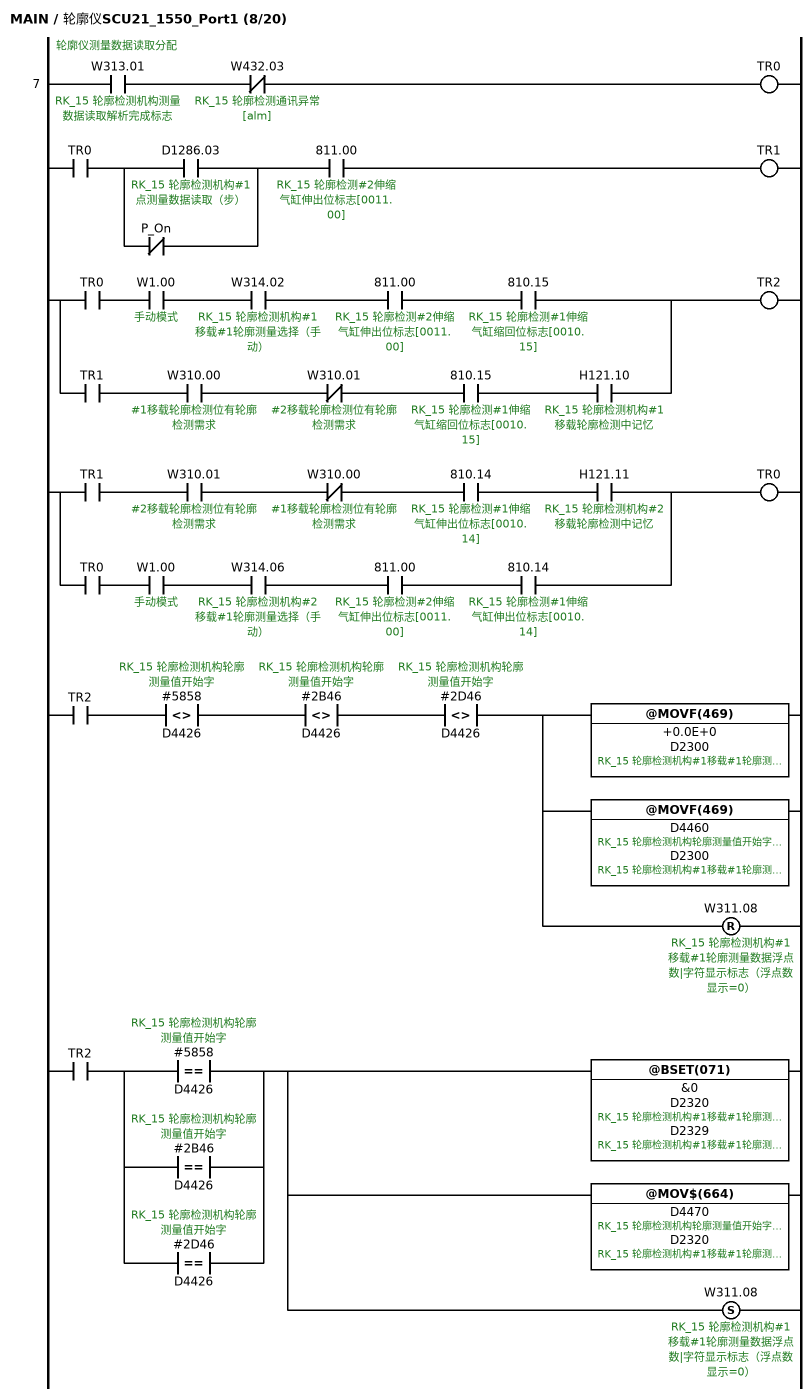
; [picture p24: MAIN / 轮廓仪SCU21_1550_Port1, rungs 7-7]

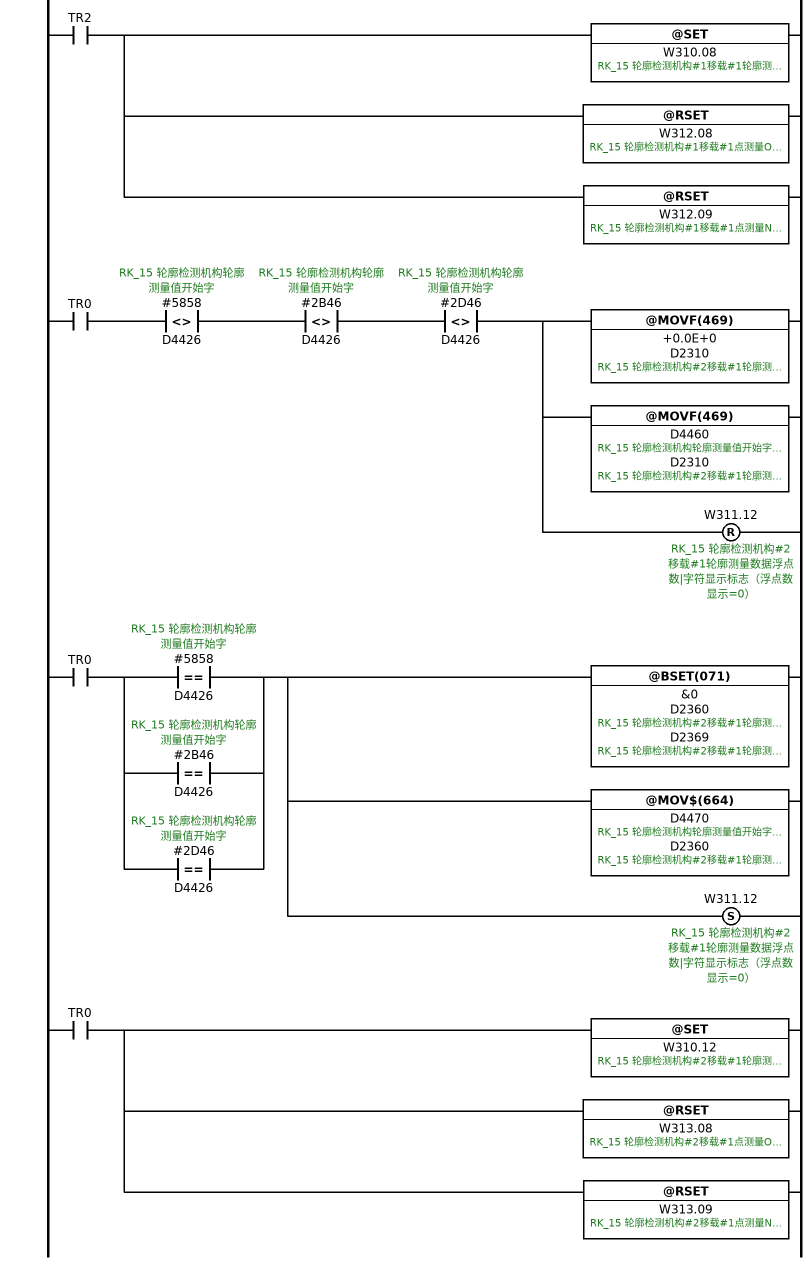
; rung 7: 轮廓仪测量数据读取分配
LD W313.01  ; RK_15 轮廓检测机构测量数据读取解析完成标志
ANDNOT W432.03  ; RK_15 轮廓检测通讯异常[alm]
OUT TR0
AND W1.00  ; 手动模式
AND W314.02  ; RK_15 轮廓检测机构#1移载#1轮廓测量选择（手动）
AND 811.00  ; RK_15 轮廓检测#2伸缩气缸伸出位标志[0011.00]
AND 810.15  ; RK_15 轮廓检测#1伸缩气缸缩回位标志[0010.15]
LD TR0
LD D1286.03  ; RK_15 轮廓检测机构#1点测量数据读取（步）
ORNOT P_On
ANDLD
AND 811.00  ; RK_15 轮廓检测#2伸缩气缸伸出位标志[0011.00]
OUT TR1
AND W310.00  ; #1移载轮廓检测位有轮廓检测需求
ANDNOT W310.01  ; #2移载轮廓检测位有轮廓检测需求
AND 810.15  ; RK_15 轮廓检测#1伸缩气缸缩回位标志[0010.15]
AND H121.10  ; RK_15 轮廓检测机构#1移载轮廓检测中记忆
ORLD
OUT TR2
AND<>(305) #5858 D4426  ; RK_15 轮廓检测机构轮廓测量值开始字
AND<>(305) #2B46 D4426  ; RK_15 轮廓检测机构轮廓测量值开始字
AND<>(305) #2D46 D4426  ; RK_15 轮廓检测机构轮廓测量值开始字
@MOVF(469) +0.0E+0 D2300  ; RK_15 轮廓检测机构#1移载#1轮廓测量值（Float）
@MOVF(469) D4460 D2300  ; RK_15 轮廓检测机构轮廓测量值开始字（Float）, RK_15 轮廓检测机构#1移载#1轮廓测量值（Float）
RSET W311.08  ; RK_15 轮廓检测机构#1移载#1轮廓测量数据浮点数|字符显示标志（浮点数显示=0）
LD TR2
LD=(300) #5858 D4426  ; RK_15 轮廓检测机构轮廓测量值开始字
OR=(300) #2B46 D4426  ; RK_15 轮廓检测机构轮廓测量值开始字
OR=(300) #2D46 D4426  ; RK_15 轮廓检测机构轮廓测量值开始字
ANDLD
@BSET(071) &0 D2320 D2329  ; RK_15 轮廓检测机构#1移载#1轮廓测量值开始字（String）, RK_15 轮廓检测机构#1移载#1轮廓测量值结束字（String）
@MOV$(664) D4470 D2320  ; RK_15 轮廓检测机构轮廓测量值开始字（String）, RK_15 轮廓检测机构#1移载#1轮廓测量值开始字（String）
SET W311.08  ; RK_15 轮廓检测机构#1移载#1轮廓测量数据浮点数|字符显示标志（浮点数显示=0）
LD TR2
@SET W310.08  ; RK_15 轮廓检测机构#1移载#1轮廓测量值读取标志
@RSET W312.08  ; RK_15 轮廓检测机构#1移载#1点测量OK标志
@RSET W312.09  ; RK_15 轮廓检测机构#1移载#1点测量NG标志
LD TR1
AND W310.01  ; #2移载轮廓检测位有轮廓检测需求
ANDNOT W310.00  ; #1移载轮廓检测位有轮廓检测需求
AND 810.14  ; RK_15 轮廓检测#1伸缩气缸伸出位标志[0010.14]
AND H121.11  ; RK_15 轮廓检测机构#2移载轮廓检测中记忆
LD TR0
AND W1.00  ; 手动模式
AND W314.06  ; RK_15 轮廓检测机构#2移载#1轮廓测量选择（手动）
AND 811.00  ; RK_15 轮廓检测#2伸缩气缸伸出位标志[0011.00]
AND 810.14  ; RK_15 轮廓检测#1伸缩气缸伸出位标志[0010.14]
ORLD
OUT TR0
AND<>(305) #5858 D4426  ; RK_15 轮廓检测机构轮廓测量值开始字
AND<>(305) #2B46 D4426  ; RK_15 轮廓检测机构轮廓测量值开始字
AND<>(305) #2D46 D4426  ; RK_15 轮廓检测机构轮廓测量值开始字
@MOVF(469) +0.0E+0 D2310  ; RK_15 轮廓检测机构#2移载#1轮廓测量值（Float）
@MOVF(469) D4460 D2310  ; RK_15 轮廓检测机构轮廓测量值开始字（Float）, RK_15 轮廓检测机构#2移载#1轮廓测量值（Float）
RSET W311.12  ; RK_15 轮廓检测机构#2移载#1轮廓测量数据浮点数|字符显示标志（浮点数显示=0）
LD TR0
LD=(300) #5858 D4426  ; RK_15 轮廓检测机构轮廓测量值开始字
OR=(300) #2B46 D4426  ; RK_15 轮廓检测机构轮廓测量值开始字
OR=(300) #2D46 D4426  ; RK_15 轮廓检测机构轮廓测量值开始字
ANDLD
@BSET(071) &0 D2360 D2369  ; RK_15 轮廓检测机构#2移载#1轮廓测量值开始字（String）, RK_15 轮廓检测机构#2移载#1轮廓测量值结束字（String）
@MOV$(664) D4470 D2360  ; RK_15 轮廓检测机构轮廓测量值开始字（String）, RK_15 轮廓检测机构#2移载#1轮廓测量值开始字（String）
SET W311.12  ; RK_15 轮廓检测机构#2移载#1轮廓测量数据浮点数|字符显示标志（浮点数显示=0）
LD TR0
@SET W310.12  ; RK_15 轮廓检测机构#2移载#1轮廓测量值读取标志
@RSET W313.08  ; RK_15 轮廓检测机构#2移载#1点测量OK标志
@RSET W313.09  ; RK_15 轮廓检测机构#2移载#1点测量NG标志

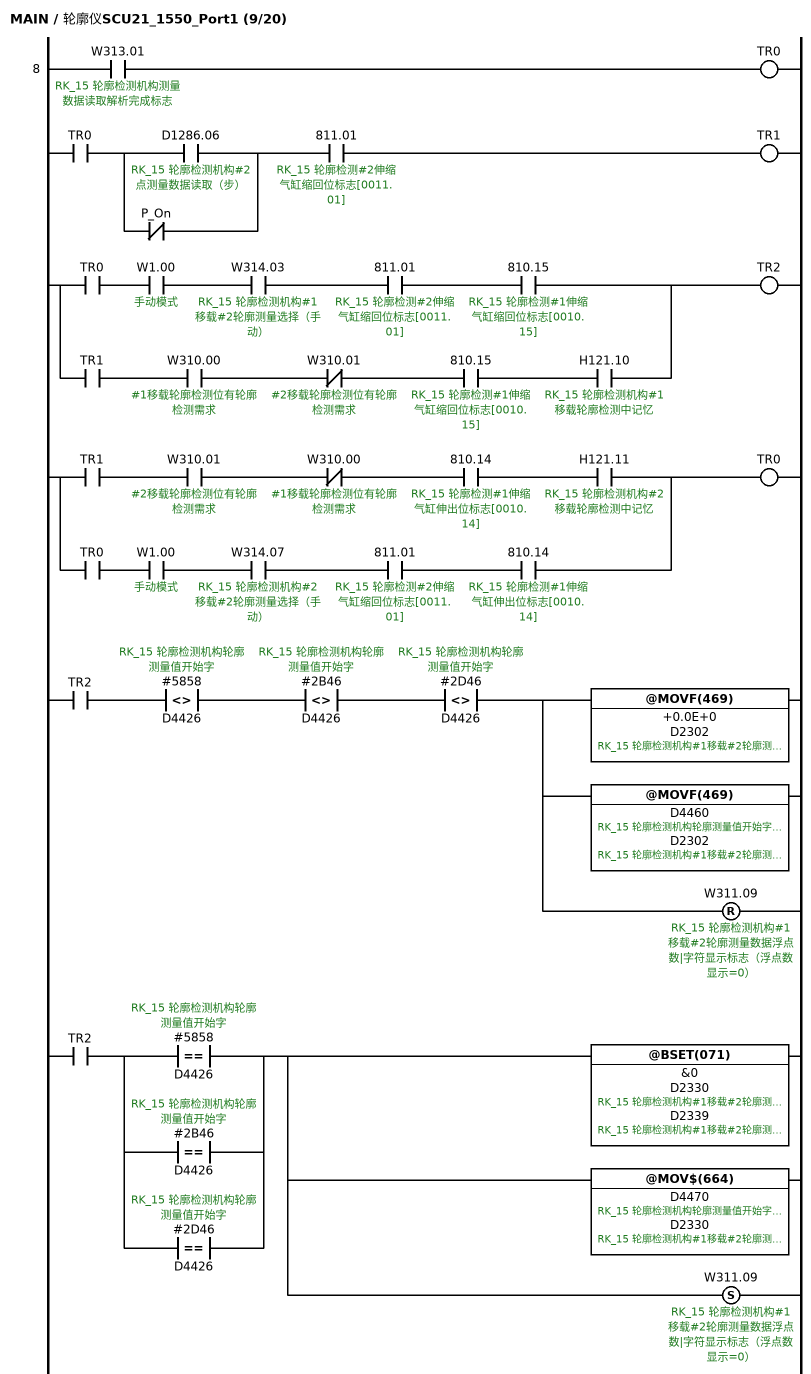

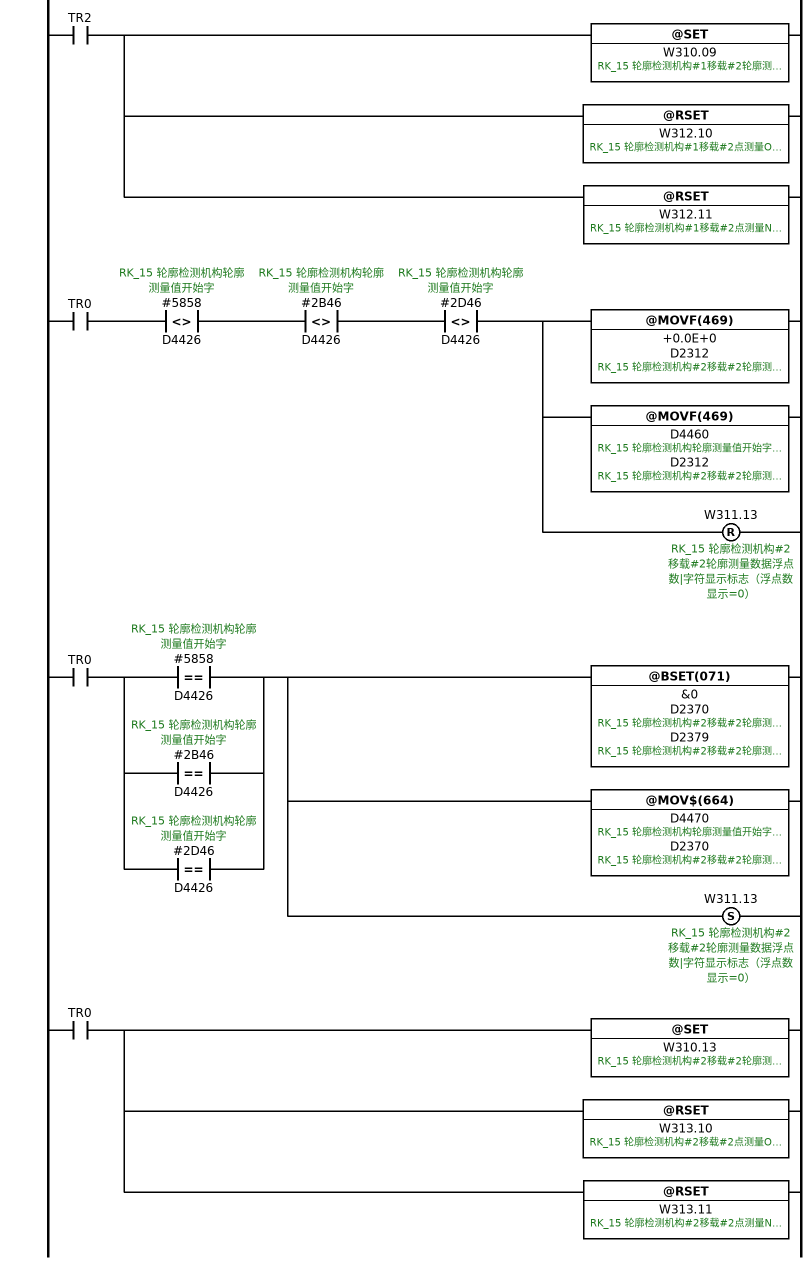
; rung 8
LD W313.01  ; RK_15 轮廓检测机构测量数据读取解析完成标志
OUT TR0
AND W1.00  ; 手动模式
AND W314.03  ; RK_15 轮廓检测机构#1移载#2轮廓测量选择（手动）
AND 811.01  ; RK_15 轮廓检测#2伸缩气缸缩回位标志[0011.01]
AND 810.15  ; RK_15 轮廓检测#1伸缩气缸缩回位标志[0010.15]
LD TR0
LD D1286.06  ; RK_15 轮廓检测机构#2点测量数据读取（步）
ORNOT P_On
ANDLD
AND 811.01  ; RK_15 轮廓检测#2伸缩气缸缩回位标志[0011.01]
OUT TR1
AND W310.00  ; #1移载轮廓检测位有轮廓检测需求
ANDNOT W310.01  ; #2移载轮廓检测位有轮廓检测需求
AND 810.15  ; RK_15 轮廓检测#1伸缩气缸缩回位标志[0010.15]
AND H121.10  ; RK_15 轮廓检测机构#1移载轮廓检测中记忆
ORLD
OUT TR2
AND<>(305) #5858 D4426  ; RK_15 轮廓检测机构轮廓测量值开始字
AND<>(305) #2B46 D4426  ; RK_15 轮廓检测机构轮廓测量值开始字
AND<>(305) #2D46 D4426  ; RK_15 轮廓检测机构轮廓测量值开始字
@MOVF(469) +0.0E+0 D2302  ; RK_15 轮廓检测机构#1移载#2轮廓测量值（Float）
@MOVF(469) D4460 D2302  ; RK_15 轮廓检测机构轮廓测量值开始字（Float）, RK_15 轮廓检测机构#1移载#2轮廓测量值（Float）
RSET W311.09  ; RK_15 轮廓检测机构#1移载#2轮廓测量数据浮点数|字符显示标志（浮点数显示=0）
LD TR2
LD=(300) #5858 D4426  ; RK_15 轮廓检测机构轮廓测量值开始字
OR=(300) #2B46 D4426  ; RK_15 轮廓检测机构轮廓测量值开始字
OR=(300) #2D46 D4426  ; RK_15 轮廓检测机构轮廓测量值开始字
ANDLD
@BSET(071) &0 D2330 D2339  ; RK_15 轮廓检测机构#1移载#2轮廓测量值开始字（String）, RK_15 轮廓检测机构#1移载#2轮廓测量值结束字（String）
@MOV$(664) D4470 D2330  ; RK_15 轮廓检测机构轮廓测量值开始字（String）, RK_15 轮廓检测机构#1移载#2轮廓测量值开始字（String）
SET W311.09  ; RK_15 轮廓检测机构#1移载#2轮廓测量数据浮点数|字符显示标志（浮点数显示=0）
LD TR2
@SET W310.09  ; RK_15 轮廓检测机构#1移载#2轮廓测量值读取标志
@RSET W312.10  ; RK_15 轮廓检测机构#1移载#2点测量OK标志
@RSET W312.11  ; RK_15 轮廓检测机构#1移载#2点测量NG标志
LD TR1
AND W310.01  ; #2移载轮廓检测位有轮廓检测需求
ANDNOT W310.00  ; #1移载轮廓检测位有轮廓检测需求
AND 810.14  ; RK_15 轮廓检测#1伸缩气缸伸出位标志[0010.14]
AND H121.11  ; RK_15 轮廓检测机构#2移载轮廓检测中记忆
LD TR0
AND W1.00  ; 手动模式
AND W314.07  ; RK_15 轮廓检测机构#2移载#2轮廓测量选择（手动）
AND 811.01  ; RK_15 轮廓检测#2伸缩气缸缩回位标志[0011.01]
AND 810.14  ; RK_15 轮廓检测#1伸缩气缸伸出位标志[0010.14]
ORLD
OUT TR0
AND<>(305) #5858 D4426  ; RK_15 轮廓检测机构轮廓测量值开始字
AND<>(305) #2B46 D4426  ; RK_15 轮廓检测机构轮廓测量值开始字
AND<>(305) #2D46 D4426  ; RK_15 轮廓检测机构轮廓测量值开始字
@MOVF(469) +0.0E+0 D2312  ; RK_15 轮廓检测机构#2移载#2轮廓测量值（Float）
@MOVF(469) D4460 D2312  ; RK_15 轮廓检测机构轮廓测量值开始字（Float）, RK_15 轮廓检测机构#2移载#2轮廓测量值（Float）
RSET W311.13  ; RK_15 轮廓检测机构#2移载#2轮廓测量数据浮点数|字符显示标志（浮点数显示=0）
LD TR0
LD=(300) #5858 D4426  ; RK_15 轮廓检测机构轮廓测量值开始字
OR=(300) #2B46 D4426  ; RK_15 轮廓检测机构轮廓测量值开始字
OR=(300) #2D46 D4426  ; RK_15 轮廓检测机构轮廓测量值开始字
ANDLD
@BSET(071) &0 D2370 D2379  ; RK_15 轮廓检测机构#2移载#2轮廓测量值开始字（String）, RK_15 轮廓检测机构#2移载#2轮廓测量值结束字（String）
@MOV$(664) D4470 D2370  ; RK_15 轮廓检测机构轮廓测量值开始字（String）, RK_15 轮廓检测机构#2移载#2轮廓测量值开始字（String）
SET W311.13  ; RK_15 轮廓检测机构#2移载#2轮廓测量数据浮点数|字符显示标志（浮点数显示=0）
LD TR0
@SET W310.13  ; RK_15 轮廓检测机构#2移载#2轮廓测量值读取标志
@RSET W313.10  ; RK_15 轮廓检测机构#2移载#2点测量OK标志
@RSET W313.11  ; RK_15 轮廓检测机构#2移载#2点测量NG标志

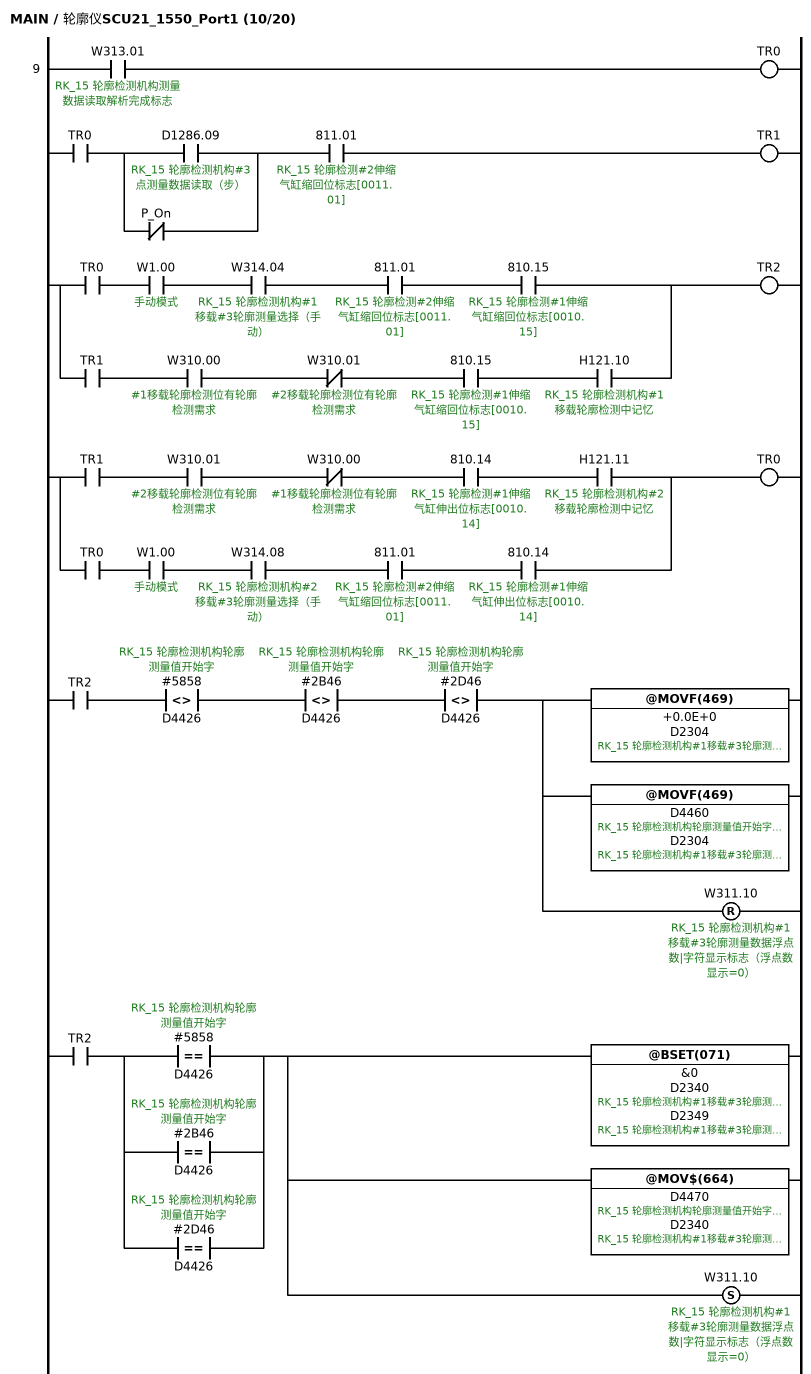

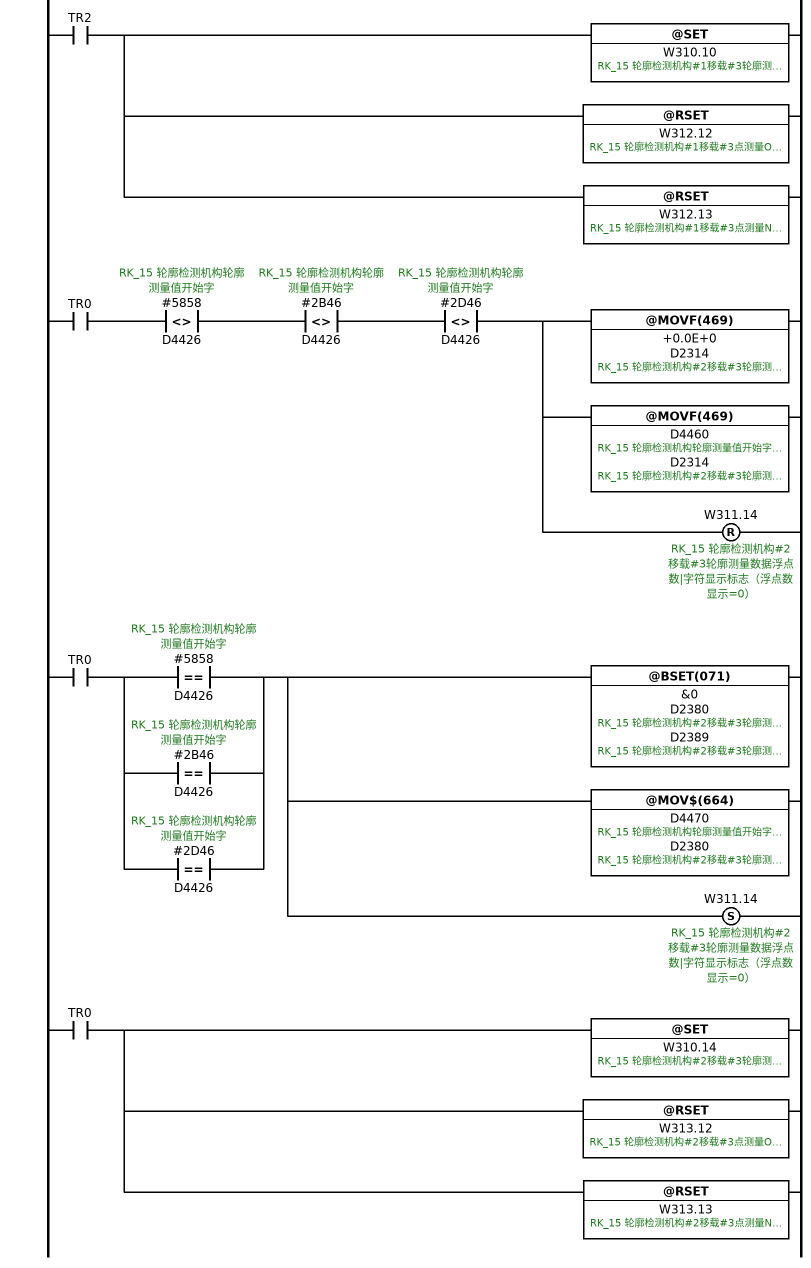
; rung 9
LD W313.01  ; RK_15 轮廓检测机构测量数据读取解析完成标志
OUT TR0
AND W1.00  ; 手动模式
AND W314.04  ; RK_15 轮廓检测机构#1移载#3轮廓测量选择（手动）
AND 811.01  ; RK_15 轮廓检测#2伸缩气缸缩回位标志[0011.01]
AND 810.15  ; RK_15 轮廓检测#1伸缩气缸缩回位标志[0010.15]
LD TR0
LD D1286.09  ; RK_15 轮廓检测机构#3点测量数据读取（步）
ORNOT P_On
ANDLD
AND 811.01  ; RK_15 轮廓检测#2伸缩气缸缩回位标志[0011.01]
OUT TR1
AND W310.00  ; #1移载轮廓检测位有轮廓检测需求
ANDNOT W310.01  ; #2移载轮廓检测位有轮廓检测需求
AND 810.15  ; RK_15 轮廓检测#1伸缩气缸缩回位标志[0010.15]
AND H121.10  ; RK_15 轮廓检测机构#1移载轮廓检测中记忆
ORLD
OUT TR2
AND<>(305) #5858 D4426  ; RK_15 轮廓检测机构轮廓测量值开始字
AND<>(305) #2B46 D4426  ; RK_15 轮廓检测机构轮廓测量值开始字
AND<>(305) #2D46 D4426  ; RK_15 轮廓检测机构轮廓测量值开始字
@MOVF(469) +0.0E+0 D2304  ; RK_15 轮廓检测机构#1移载#3轮廓测量值（Float）
@MOVF(469) D4460 D2304  ; RK_15 轮廓检测机构轮廓测量值开始字（Float）, RK_15 轮廓检测机构#1移载#3轮廓测量值（Float）
RSET W311.10  ; RK_15 轮廓检测机构#1移载#3轮廓测量数据浮点数|字符显示标志（浮点数显示=0）
LD TR2
LD=(300) #5858 D4426  ; RK_15 轮廓检测机构轮廓测量值开始字
OR=(300) #2B46 D4426  ; RK_15 轮廓检测机构轮廓测量值开始字
OR=(300) #2D46 D4426  ; RK_15 轮廓检测机构轮廓测量值开始字
ANDLD
@BSET(071) &0 D2340 D2349  ; RK_15 轮廓检测机构#1移载#3轮廓测量值开始字（String）, RK_15 轮廓检测机构#1移载#3轮廓测量值结束字（String）
@MOV$(664) D4470 D2340  ; RK_15 轮廓检测机构轮廓测量值开始字（String）, RK_15 轮廓检测机构#1移载#3轮廓测量值开始字（String）
SET W311.10  ; RK_15 轮廓检测机构#1移载#3轮廓测量数据浮点数|字符显示标志（浮点数显示=0）
LD TR2
@SET W310.10  ; RK_15 轮廓检测机构#1移载#3轮廓测量值读取标志
@RSET W312.12  ; RK_15 轮廓检测机构#1移载#3点测量OK标志
@RSET W312.13  ; RK_15 轮廓检测机构#1移载#3点测量NG标志
LD TR1
AND W310.01  ; #2移载轮廓检测位有轮廓检测需求
ANDNOT W310.00  ; #1移载轮廓检测位有轮廓检测需求
AND 810.14  ; RK_15 轮廓检测#1伸缩气缸伸出位标志[0010.14]
AND H121.11  ; RK_15 轮廓检测机构#2移载轮廓检测中记忆
LD TR0
AND W1.00  ; 手动模式
AND W314.08  ; RK_15 轮廓检测机构#2移载#3轮廓测量选择（手动）
AND 811.01  ; RK_15 轮廓检测#2伸缩气缸缩回位标志[0011.01]
AND 810.14  ; RK_15 轮廓检测#1伸缩气缸伸出位标志[0010.14]
ORLD
OUT TR0
AND<>(305) #5858 D4426  ; RK_15 轮廓检测机构轮廓测量值开始字
AND<>(305) #2B46 D4426  ; RK_15 轮廓检测机构轮廓测量值开始字
AND<>(305) #2D46 D4426  ; RK_15 轮廓检测机构轮廓测量值开始字
@MOVF(469) +0.0E+0 D2314  ; RK_15 轮廓检测机构#2移载#3轮廓测量值（Float）
@MOVF(469) D4460 D2314  ; RK_15 轮廓检测机构轮廓测量值开始字（Float）, RK_15 轮廓检测机构#2移载#3轮廓测量值（Float）
RSET W311.14  ; RK_15 轮廓检测机构#2移载#3轮廓测量数据浮点数|字符显示标志（浮点数显示=0）
LD TR0
LD=(300) #5858 D4426  ; RK_15 轮廓检测机构轮廓测量值开始字
OR=(300) #2B46 D4426  ; RK_15 轮廓检测机构轮廓测量值开始字
OR=(300) #2D46 D4426  ; RK_15 轮廓检测机构轮廓测量值开始字
ANDLD
@BSET(071) &0 D2380 D2389  ; RK_15 轮廓检测机构#2移载#3轮廓测量值开始字（String）, RK_15 轮廓检测机构#2移载#3轮廓测量值结束字（String）
@MOV$(664) D4470 D2380  ; RK_15 轮廓检测机构轮廓测量值开始字（String）, RK_15 轮廓检测机构#2移载#3轮廓测量值开始字（String）
SET W311.14  ; RK_15 轮廓检测机构#2移载#3轮廓测量数据浮点数|字符显示标志（浮点数显示=0）
LD TR0
@SET W310.14  ; RK_15 轮廓检测机构#2移载#3轮廓测量值读取标志
@RSET W313.12  ; RK_15 轮廓检测机构#2移载#3点测量OK标志
@RSET W313.13  ; RK_15 轮廓检测机构#2移载#3点测量NG标志

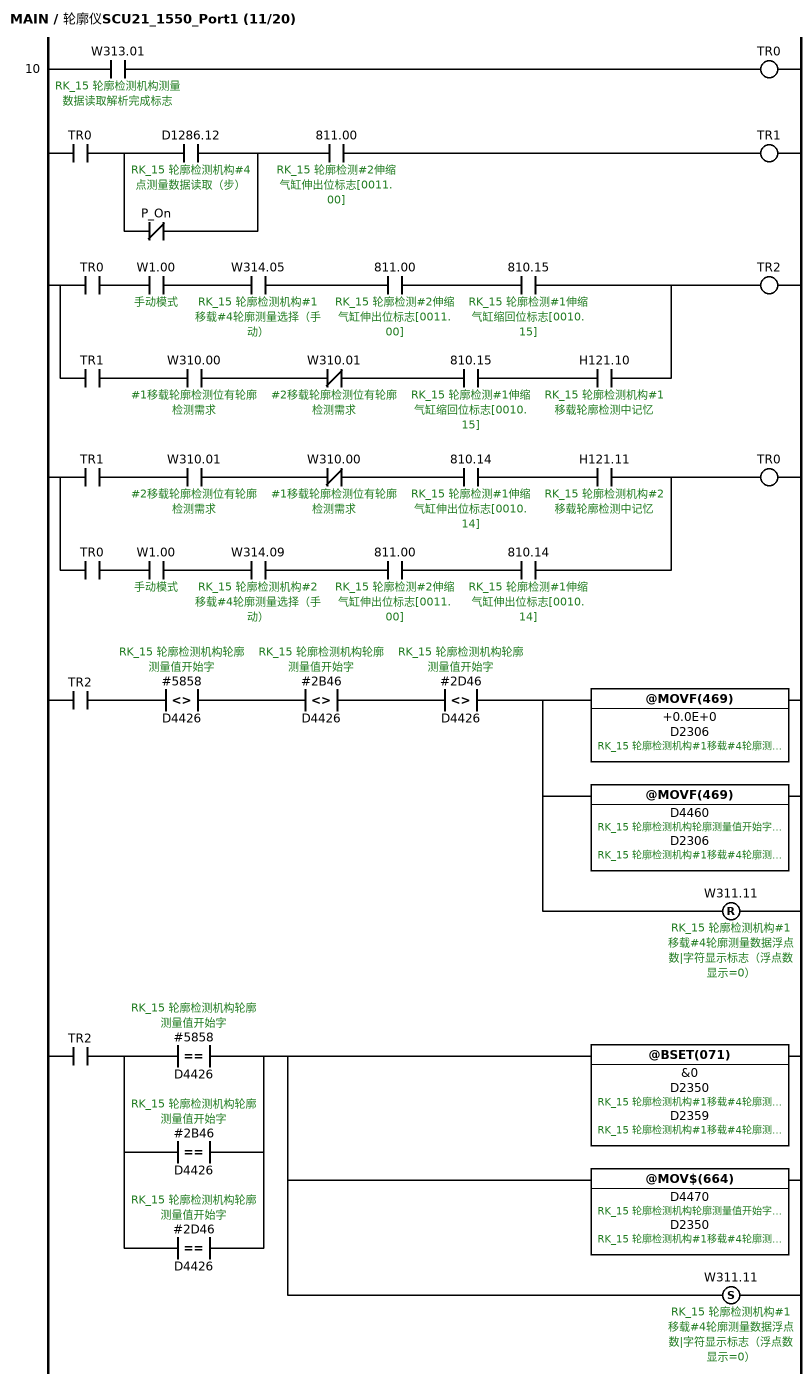

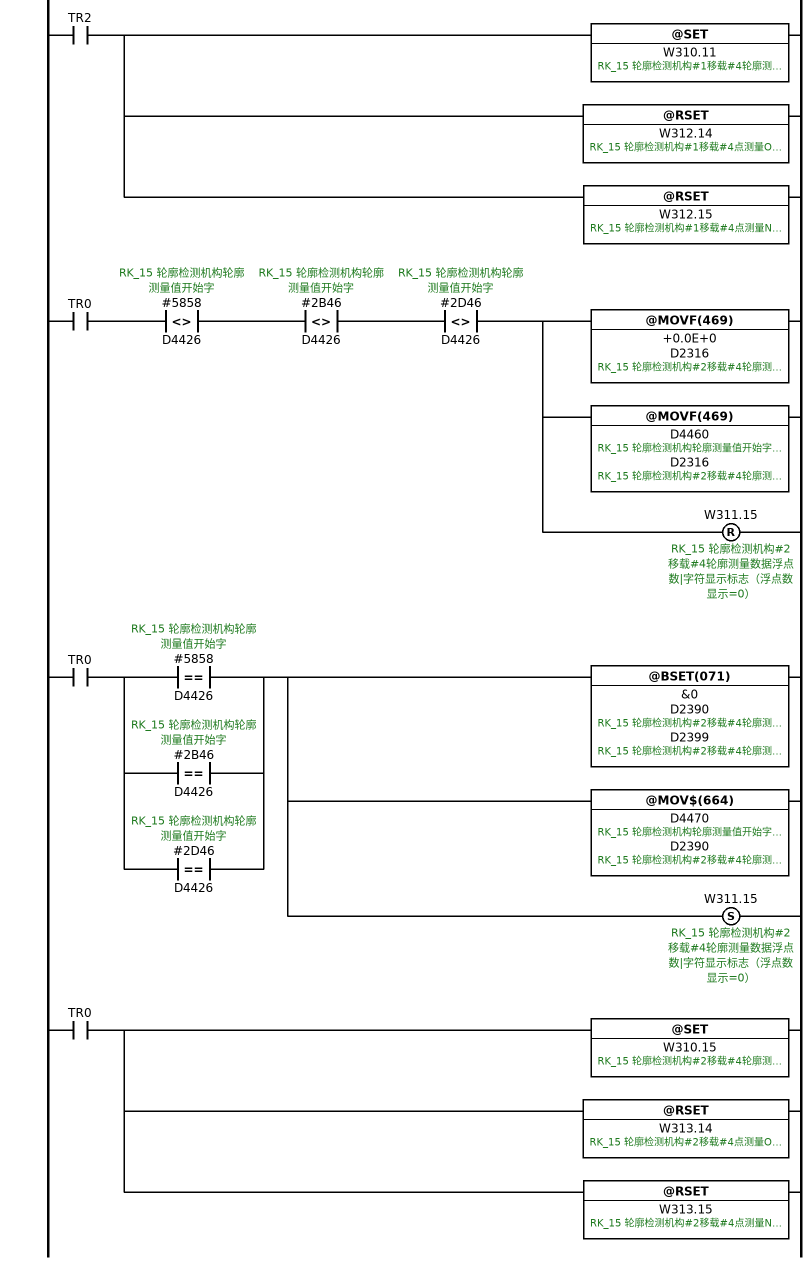
; rung 10
LD W313.01  ; RK_15 轮廓检测机构测量数据读取解析完成标志
OUT TR0
AND W1.00  ; 手动模式
AND W314.05  ; RK_15 轮廓检测机构#1移载#4轮廓测量选择（手动）
AND 811.00  ; RK_15 轮廓检测#2伸缩气缸伸出位标志[0011.00]
AND 810.15  ; RK_15 轮廓检测#1伸缩气缸缩回位标志[0010.15]
LD TR0
LD D1286.12  ; RK_15 轮廓检测机构#4点测量数据读取（步）
ORNOT P_On
ANDLD
AND 811.00  ; RK_15 轮廓检测#2伸缩气缸伸出位标志[0011.00]
OUT TR1
AND W310.00  ; #1移载轮廓检测位有轮廓检测需求
ANDNOT W310.01  ; #2移载轮廓检测位有轮廓检测需求
AND 810.15  ; RK_15 轮廓检测#1伸缩气缸缩回位标志[0010.15]
AND H121.10  ; RK_15 轮廓检测机构#1移载轮廓检测中记忆
ORLD
OUT TR2
AND<>(305) #5858 D4426  ; RK_15 轮廓检测机构轮廓测量值开始字
AND<>(305) #2B46 D4426  ; RK_15 轮廓检测机构轮廓测量值开始字
AND<>(305) #2D46 D4426  ; RK_15 轮廓检测机构轮廓测量值开始字
@MOVF(469) +0.0E+0 D2306  ; RK_15 轮廓检测机构#1移载#4轮廓测量值（Float）
@MOVF(469) D4460 D2306  ; RK_15 轮廓检测机构轮廓测量值开始字（Float）, RK_15 轮廓检测机构#1移载#4轮廓测量值（Float）
RSET W311.11  ; RK_15 轮廓检测机构#1移载#4轮廓测量数据浮点数|字符显示标志（浮点数显示=0）
LD TR2
LD=(300) #5858 D4426  ; RK_15 轮廓检测机构轮廓测量值开始字
OR=(300) #2B46 D4426  ; RK_15 轮廓检测机构轮廓测量值开始字
OR=(300) #2D46 D4426  ; RK_15 轮廓检测机构轮廓测量值开始字
ANDLD
@BSET(071) &0 D2350 D2359  ; RK_15 轮廓检测机构#1移载#4轮廓测量值开始字（String）, RK_15 轮廓检测机构#1移载#4轮廓测量值结束字（String）
@MOV$(664) D4470 D2350  ; RK_15 轮廓检测机构轮廓测量值开始字（String）, RK_15 轮廓检测机构#1移载#4轮廓测量值开始字（String）
SET W311.11  ; RK_15 轮廓检测机构#1移载#4轮廓测量数据浮点数|字符显示标志（浮点数显示=0）
LD TR2
@SET W310.11  ; RK_15 轮廓检测机构#1移载#4轮廓测量值读取标志
@RSET W312.14  ; RK_15 轮廓检测机构#1移载#4点测量OK标志
@RSET W312.15  ; RK_15 轮廓检测机构#1移载#4点测量NG标志
LD TR1
AND W310.01  ; #2移载轮廓检测位有轮廓检测需求
ANDNOT W310.00  ; #1移载轮廓检测位有轮廓检测需求
AND 810.14  ; RK_15 轮廓检测#1伸缩气缸伸出位标志[0010.14]
AND H121.11  ; RK_15 轮廓检测机构#2移载轮廓检测中记忆
LD TR0
AND W1.00  ; 手动模式
AND W314.09  ; RK_15 轮廓检测机构#2移载#4轮廓测量选择（手动）
AND 811.00  ; RK_15 轮廓检测#2伸缩气缸伸出位标志[0011.00]
AND 810.14  ; RK_15 轮廓检测#1伸缩气缸伸出位标志[0010.14]
ORLD
OUT TR0
AND<>(305) #5858 D4426  ; RK_15 轮廓检测机构轮廓测量值开始字
AND<>(305) #2B46 D4426  ; RK_15 轮廓检测机构轮廓测量值开始字
AND<>(305) #2D46 D4426  ; RK_15 轮廓检测机构轮廓测量值开始字
@MOVF(469) +0.0E+0 D2316  ; RK_15 轮廓检测机构#2移载#4轮廓测量值（Float）
@MOVF(469) D4460 D2316  ; RK_15 轮廓检测机构轮廓测量值开始字（Float）, RK_15 轮廓检测机构#2移载#4轮廓测量值（Float）
RSET W311.15  ; RK_15 轮廓检测机构#2移载#4轮廓测量数据浮点数|字符显示标志（浮点数显示=0）
LD TR0
LD=(300) #5858 D4426  ; RK_15 轮廓检测机构轮廓测量值开始字
OR=(300) #2B46 D4426  ; RK_15 轮廓检测机构轮廓测量值开始字
OR=(300) #2D46 D4426  ; RK_15 轮廓检测机构轮廓测量值开始字
ANDLD
@BSET(071) &0 D2390 D2399  ; RK_15 轮廓检测机构#2移载#4轮廓测量值开始字（String）, RK_15 轮廓检测机构#2移载#4轮廓测量值结束字（String）
@MOV$(664) D4470 D2390  ; RK_15 轮廓检测机构轮廓测量值开始字（String）, RK_15 轮廓检测机构#2移载#4轮廓测量值开始字（String）
SET W311.15  ; RK_15 轮廓检测机构#2移载#4轮廓测量数据浮点数|字符显示标志（浮点数显示=0）
LD TR0
@SET W310.15  ; RK_15 轮廓检测机构#2移载#4轮廓测量值读取标志
@RSET W313.14  ; RK_15 轮廓检测机构#2移载#4点测量OK标志
@RSET W313.15  ; RK_15 轮廓检测机构#2移载#4点测量NG标志

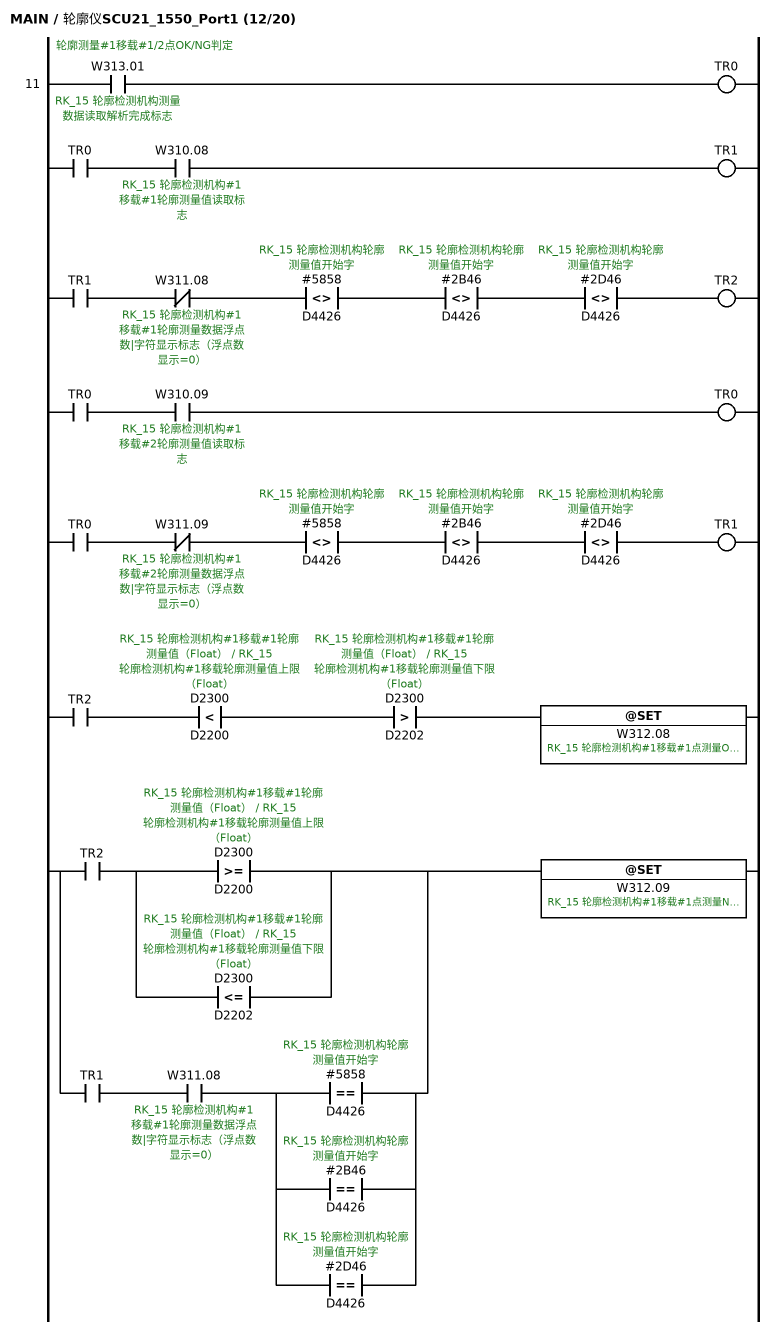

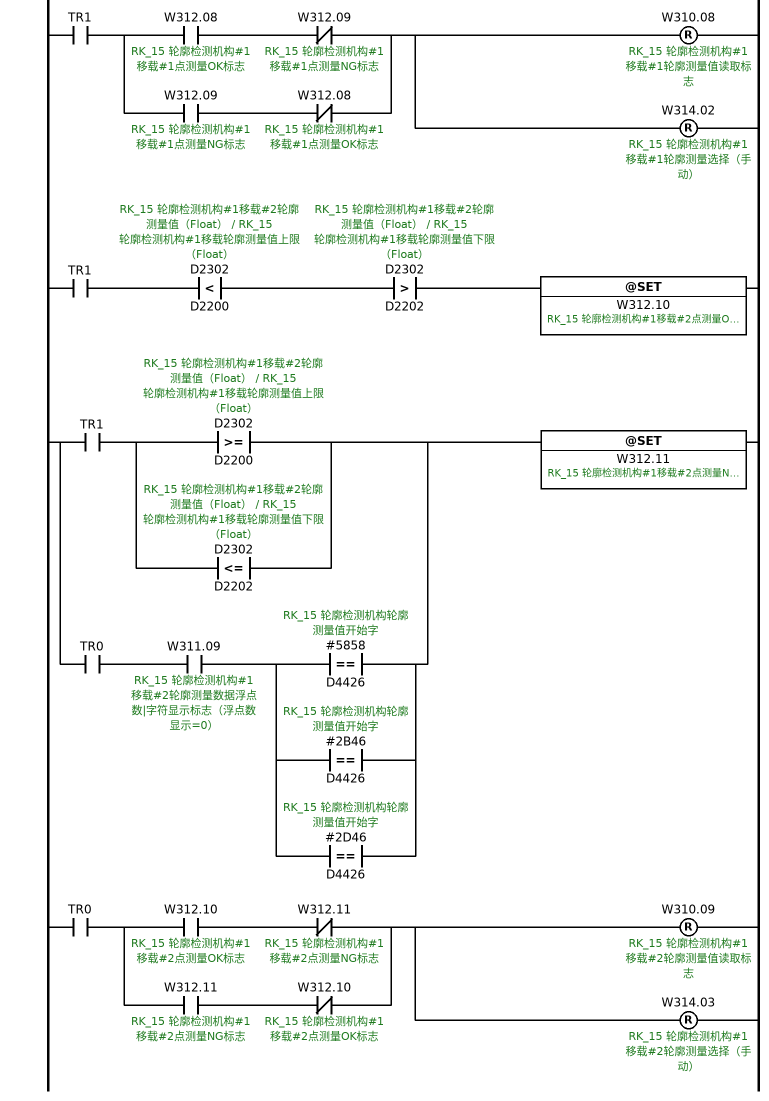
; rung 11: 轮廓测量#1移载#1/2点OK/NG判定
LD W313.01  ; RK_15 轮廓检测机构测量数据读取解析完成标志
OUT TR0
AND W310.08  ; RK_15 轮廓检测机构#1移载#1轮廓测量值读取标志
OUT TR1
ANDNOT W311.08  ; RK_15 轮廓检测机构#1移载#1轮廓测量数据浮点数|字符显示标志（浮点数显示=0）
AND<>(305) #5858 D4426  ; RK_15 轮廓检测机构轮廓测量值开始字
AND<>(305) #2B46 D4426  ; RK_15 轮廓检测机构轮廓测量值开始字
AND<>(305) #2D46 D4426  ; RK_15 轮廓检测机构轮廓测量值开始字
OUT TR2
AND<F(331) D2300 D2200  ; RK_15 轮廓检测机构#1移载#1轮廓测量值（Float）, RK_15 轮廓检测机构#1移载轮廓测量值上限（Float）
AND>F(333) D2300 D2202  ; RK_15 轮廓检测机构#1移载#1轮廓测量值（Float）, RK_15 轮廓检测机构#1移载轮廓测量值下限（Float）
@SET W312.08  ; RK_15 轮廓检测机构#1移载#1点测量OK标志
LD TR2
LD>=F(334) D2300 D2200  ; RK_15 轮廓检测机构#1移载#1轮廓测量值（Float）, RK_15 轮廓检测机构#1移载轮廓测量值上限（Float）
OR<=F(332) D2300 D2202  ; RK_15 轮廓检测机构#1移载#1轮廓测量值（Float）, RK_15 轮廓检测机构#1移载轮廓测量值下限（Float）
ANDLD
LD TR1
AND W311.08  ; RK_15 轮廓检测机构#1移载#1轮廓测量数据浮点数|字符显示标志（浮点数显示=0）
LD=(300) #5858 D4426  ; RK_15 轮廓检测机构轮廓测量值开始字
OR=(300) #2B46 D4426  ; RK_15 轮廓检测机构轮廓测量值开始字
OR=(300) #2D46 D4426  ; RK_15 轮廓检测机构轮廓测量值开始字
ANDLD
ORLD
@SET W312.09  ; RK_15 轮廓检测机构#1移载#1点测量NG标志
LD TR1
LD W312.08  ; RK_15 轮廓检测机构#1移载#1点测量OK标志
ANDNOT W312.09  ; RK_15 轮廓检测机构#1移载#1点测量NG标志
LD W312.09  ; RK_15 轮廓检测机构#1移载#1点测量NG标志
ANDNOT W312.08  ; RK_15 轮廓检测机构#1移载#1点测量OK标志
ORLD
ANDLD
RSET W310.08  ; RK_15 轮廓检测机构#1移载#1轮廓测量值读取标志
RSET W314.02  ; RK_15 轮廓检测机构#1移载#1轮廓测量选择（手动）
LD TR0
AND W310.09  ; RK_15 轮廓检测机构#1移载#2轮廓测量值读取标志
OUT TR0
ANDNOT W311.09  ; RK_15 轮廓检测机构#1移载#2轮廓测量数据浮点数|字符显示标志（浮点数显示=0）
AND<>(305) #5858 D4426  ; RK_15 轮廓检测机构轮廓测量值开始字
AND<>(305) #2B46 D4426  ; RK_15 轮廓检测机构轮廓测量值开始字
AND<>(305) #2D46 D4426  ; RK_15 轮廓检测机构轮廓测量值开始字
OUT TR1
AND<F(331) D2302 D2200  ; RK_15 轮廓检测机构#1移载#2轮廓测量值（Float）, RK_15 轮廓检测机构#1移载轮廓测量值上限（Float）
AND>F(333) D2302 D2202  ; RK_15 轮廓检测机构#1移载#2轮廓测量值（Float）, RK_15 轮廓检测机构#1移载轮廓测量值下限（Float）
@SET W312.10  ; RK_15 轮廓检测机构#1移载#2点测量OK标志
LD TR1
LD>=F(334) D2302 D2200  ; RK_15 轮廓检测机构#1移载#2轮廓测量值（Float）, RK_15 轮廓检测机构#1移载轮廓测量值上限（Float）
OR<=F(332) D2302 D2202  ; RK_15 轮廓检测机构#1移载#2轮廓测量值（Float）, RK_15 轮廓检测机构#1移载轮廓测量值下限（Float）
ANDLD
LD TR0
AND W311.09  ; RK_15 轮廓检测机构#1移载#2轮廓测量数据浮点数|字符显示标志（浮点数显示=0）
LD=(300) #5858 D4426  ; RK_15 轮廓检测机构轮廓测量值开始字
OR=(300) #2B46 D4426  ; RK_15 轮廓检测机构轮廓测量值开始字
OR=(300) #2D46 D4426  ; RK_15 轮廓检测机构轮廓测量值开始字
ANDLD
ORLD
@SET W312.11  ; RK_15 轮廓检测机构#1移载#2点测量NG标志
LD TR0
LD W312.10  ; RK_15 轮廓检测机构#1移载#2点测量OK标志
ANDNOT W312.11  ; RK_15 轮廓检测机构#1移载#2点测量NG标志
LD W312.11  ; RK_15 轮廓检测机构#1移载#2点测量NG标志
ANDNOT W312.10  ; RK_15 轮廓检测机构#1移载#2点测量OK标志
ORLD
ANDLD
RSET W310.09  ; RK_15 轮廓检测机构#1移载#2轮廓测量值读取标志
RSET W314.03  ; RK_15 轮廓检测机构#1移载#2轮廓测量选择（手动）

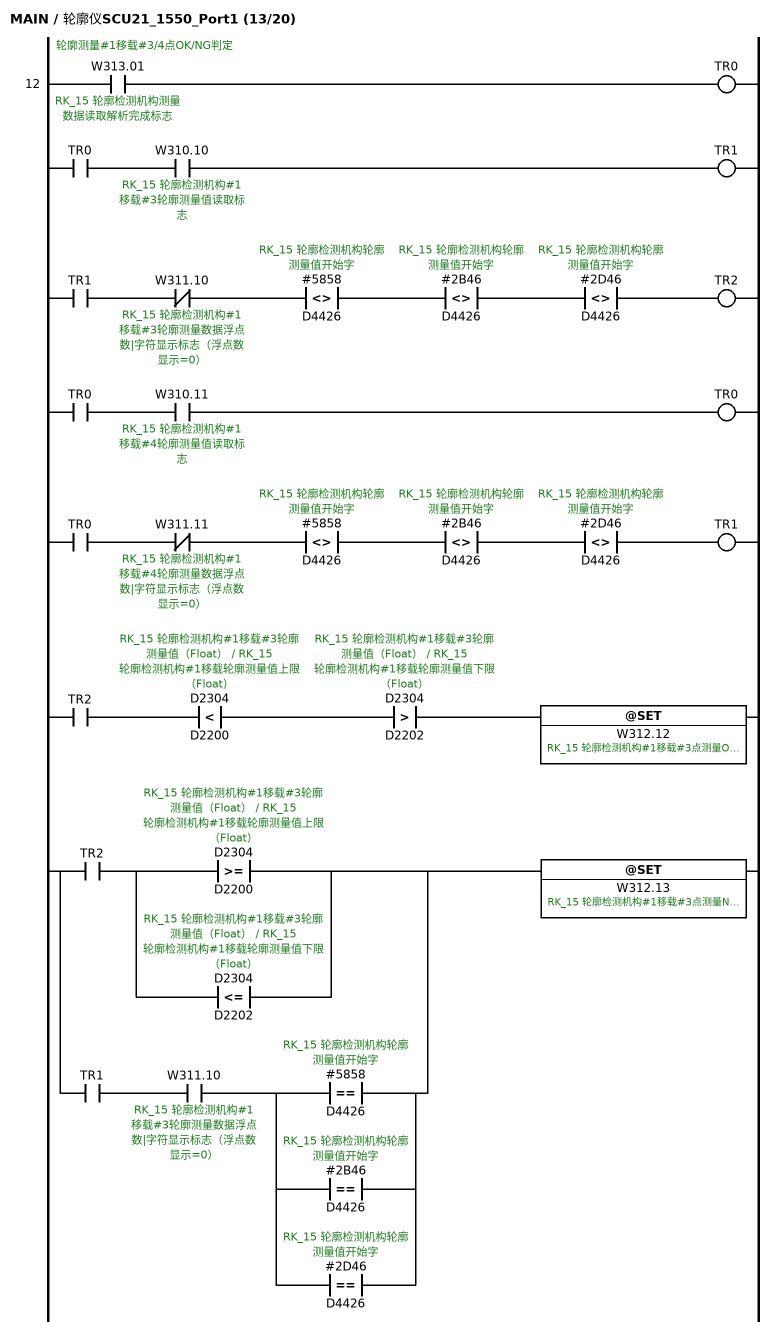

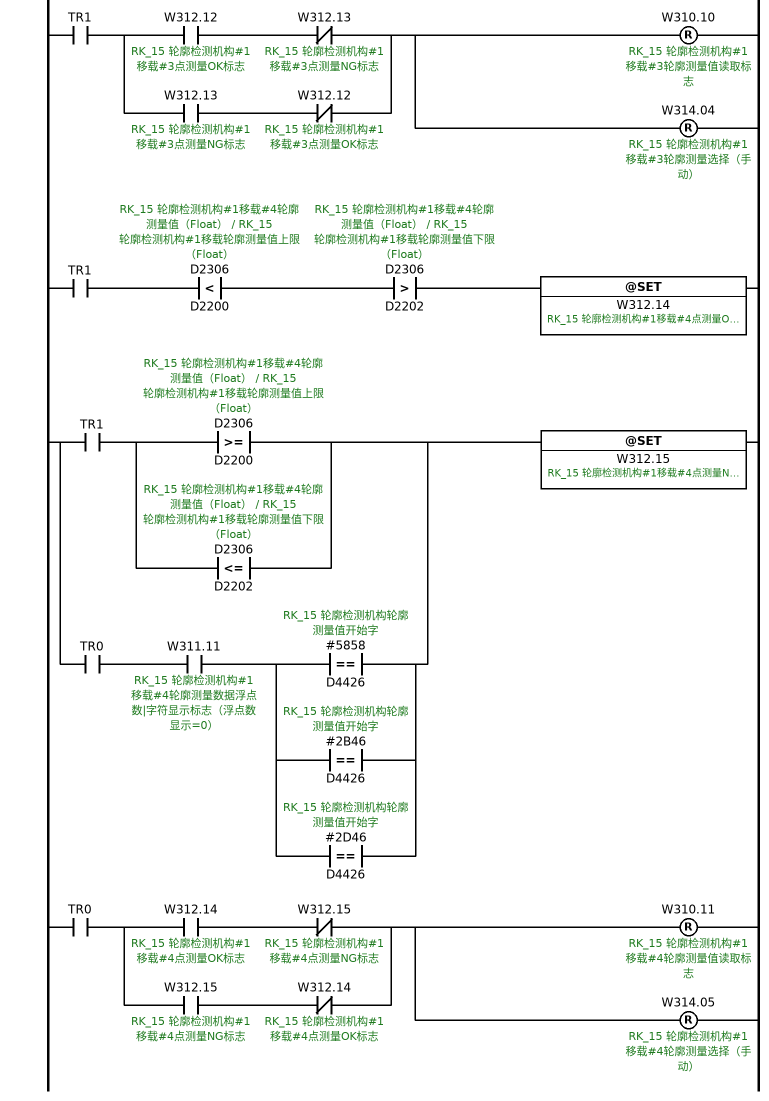
; rung 12: 轮廓测量#1移载#3/4点OK/NG判定
LD W313.01  ; RK_15 轮廓检测机构测量数据读取解析完成标志
OUT TR0
AND W310.10  ; RK_15 轮廓检测机构#1移载#3轮廓测量值读取标志
OUT TR1
ANDNOT W311.10  ; RK_15 轮廓检测机构#1移载#3轮廓测量数据浮点数|字符显示标志（浮点数显示=0）
AND<>(305) #5858 D4426  ; RK_15 轮廓检测机构轮廓测量值开始字
AND<>(305) #2B46 D4426  ; RK_15 轮廓检测机构轮廓测量值开始字
AND<>(305) #2D46 D4426  ; RK_15 轮廓检测机构轮廓测量值开始字
OUT TR2
AND<F(331) D2304 D2200  ; RK_15 轮廓检测机构#1移载#3轮廓测量值（Float）, RK_15 轮廓检测机构#1移载轮廓测量值上限（Float）
AND>F(333) D2304 D2202  ; RK_15 轮廓检测机构#1移载#3轮廓测量值（Float）, RK_15 轮廓检测机构#1移载轮廓测量值下限（Float）
@SET W312.12  ; RK_15 轮廓检测机构#1移载#3点测量OK标志
LD TR2
LD>=F(334) D2304 D2200  ; RK_15 轮廓检测机构#1移载#3轮廓测量值（Float）, RK_15 轮廓检测机构#1移载轮廓测量值上限（Float）
OR<=F(332) D2304 D2202  ; RK_15 轮廓检测机构#1移载#3轮廓测量值（Float）, RK_15 轮廓检测机构#1移载轮廓测量值下限（Float）
ANDLD
LD TR1
AND W311.10  ; RK_15 轮廓检测机构#1移载#3轮廓测量数据浮点数|字符显示标志（浮点数显示=0）
LD=(300) #5858 D4426  ; RK_15 轮廓检测机构轮廓测量值开始字
OR=(300) #2B46 D4426  ; RK_15 轮廓检测机构轮廓测量值开始字
OR=(300) #2D46 D4426  ; RK_15 轮廓检测机构轮廓测量值开始字
ANDLD
ORLD
@SET W312.13  ; RK_15 轮廓检测机构#1移载#3点测量NG标志
LD TR1
LD W312.12  ; RK_15 轮廓检测机构#1移载#3点测量OK标志
ANDNOT W312.13  ; RK_15 轮廓检测机构#1移载#3点测量NG标志
LD W312.13  ; RK_15 轮廓检测机构#1移载#3点测量NG标志
ANDNOT W312.12  ; RK_15 轮廓检测机构#1移载#3点测量OK标志
ORLD
ANDLD
RSET W310.10  ; RK_15 轮廓检测机构#1移载#3轮廓测量值读取标志
RSET W314.04  ; RK_15 轮廓检测机构#1移载#3轮廓测量选择（手动）
LD TR0
AND W310.11  ; RK_15 轮廓检测机构#1移载#4轮廓测量值读取标志
OUT TR0
ANDNOT W311.11  ; RK_15 轮廓检测机构#1移载#4轮廓测量数据浮点数|字符显示标志（浮点数显示=0）
AND<>(305) #5858 D4426  ; RK_15 轮廓检测机构轮廓测量值开始字
AND<>(305) #2B46 D4426  ; RK_15 轮廓检测机构轮廓测量值开始字
AND<>(305) #2D46 D4426  ; RK_15 轮廓检测机构轮廓测量值开始字
OUT TR1
AND<F(331) D2306 D2200  ; RK_15 轮廓检测机构#1移载#4轮廓测量值（Float）, RK_15 轮廓检测机构#1移载轮廓测量值上限（Float）
AND>F(333) D2306 D2202  ; RK_15 轮廓检测机构#1移载#4轮廓测量值（Float）, RK_15 轮廓检测机构#1移载轮廓测量值下限（Float）
@SET W312.14  ; RK_15 轮廓检测机构#1移载#4点测量OK标志
LD TR1
LD>=F(334) D2306 D2200  ; RK_15 轮廓检测机构#1移载#4轮廓测量值（Float）, RK_15 轮廓检测机构#1移载轮廓测量值上限（Float）
OR<=F(332) D2306 D2202  ; RK_15 轮廓检测机构#1移载#4轮廓测量值（Float）, RK_15 轮廓检测机构#1移载轮廓测量值下限（Float）
ANDLD
LD TR0
AND W311.11  ; RK_15 轮廓检测机构#1移载#4轮廓测量数据浮点数|字符显示标志（浮点数显示=0）
LD=(300) #5858 D4426  ; RK_15 轮廓检测机构轮廓测量值开始字
OR=(300) #2B46 D4426  ; RK_15 轮廓检测机构轮廓测量值开始字
OR=(300) #2D46 D4426  ; RK_15 轮廓检测机构轮廓测量值开始字
ANDLD
ORLD
@SET W312.15  ; RK_15 轮廓检测机构#1移载#4点测量NG标志
LD TR0
LD W312.14  ; RK_15 轮廓检测机构#1移载#4点测量OK标志
ANDNOT W312.15  ; RK_15 轮廓检测机构#1移载#4点测量NG标志
LD W312.15  ; RK_15 轮廓检测机构#1移载#4点测量NG标志
ANDNOT W312.14  ; RK_15 轮廓检测机构#1移载#4点测量OK标志
ORLD
ANDLD
RSET W310.11  ; RK_15 轮廓检测机构#1移载#4轮廓测量值读取标志
RSET W314.05  ; RK_15 轮廓检测机构#1移载#4轮廓测量选择（手动）

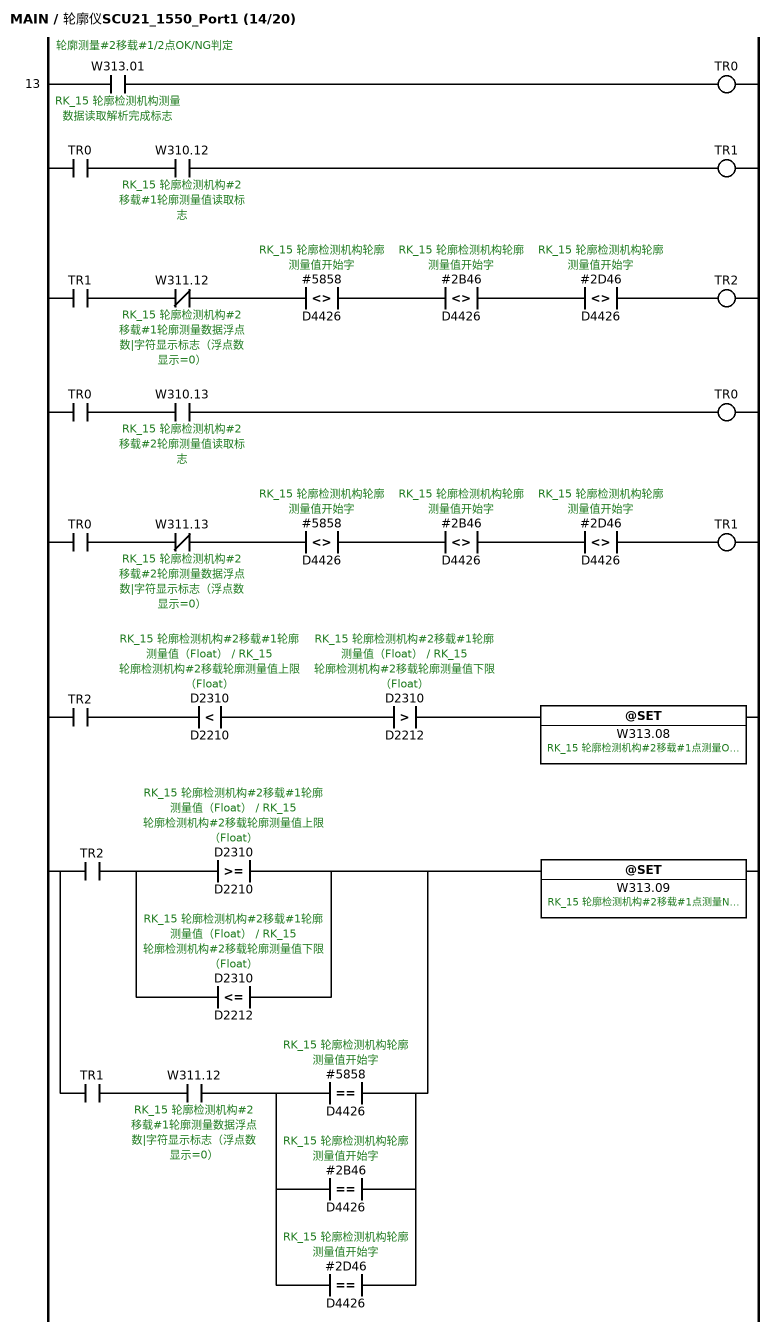

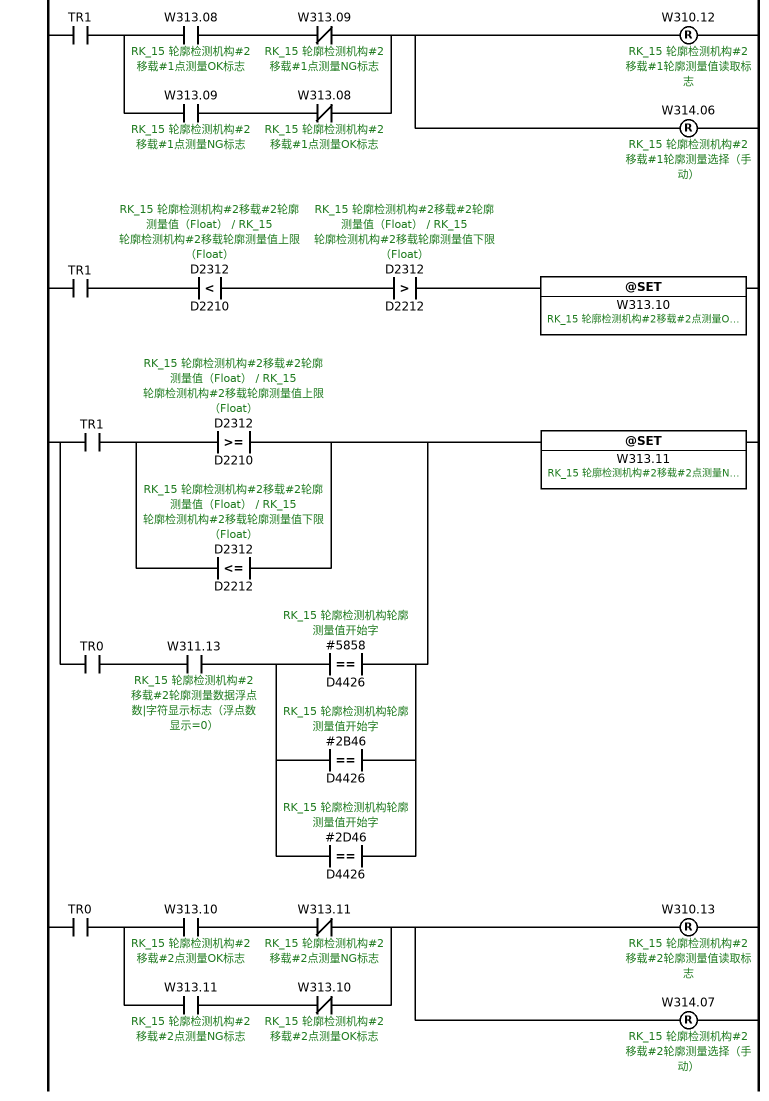
; rung 13: 轮廓测量#2移载#1/2点OK/NG判定
LD W313.01  ; RK_15 轮廓检测机构测量数据读取解析完成标志
OUT TR0
AND W310.12  ; RK_15 轮廓检测机构#2移载#1轮廓测量值读取标志
OUT TR1
ANDNOT W311.12  ; RK_15 轮廓检测机构#2移载#1轮廓测量数据浮点数|字符显示标志（浮点数显示=0）
AND<>(305) #5858 D4426  ; RK_15 轮廓检测机构轮廓测量值开始字
AND<>(305) #2B46 D4426  ; RK_15 轮廓检测机构轮廓测量值开始字
AND<>(305) #2D46 D4426  ; RK_15 轮廓检测机构轮廓测量值开始字
OUT TR2
AND<F(331) D2310 D2210  ; RK_15 轮廓检测机构#2移载#1轮廓测量值（Float）, RK_15 轮廓检测机构#2移载轮廓测量值上限（Float）
AND>F(333) D2310 D2212  ; RK_15 轮廓检测机构#2移载#1轮廓测量值（Float）, RK_15 轮廓检测机构#2移载轮廓测量值下限（Float）
@SET W313.08  ; RK_15 轮廓检测机构#2移载#1点测量OK标志
LD TR2
LD>=F(334) D2310 D2210  ; RK_15 轮廓检测机构#2移载#1轮廓测量值（Float）, RK_15 轮廓检测机构#2移载轮廓测量值上限（Float）
OR<=F(332) D2310 D2212  ; RK_15 轮廓检测机构#2移载#1轮廓测量值（Float）, RK_15 轮廓检测机构#2移载轮廓测量值下限（Float）
ANDLD
LD TR1
AND W311.12  ; RK_15 轮廓检测机构#2移载#1轮廓测量数据浮点数|字符显示标志（浮点数显示=0）
LD=(300) #5858 D4426  ; RK_15 轮廓检测机构轮廓测量值开始字
OR=(300) #2B46 D4426  ; RK_15 轮廓检测机构轮廓测量值开始字
OR=(300) #2D46 D4426  ; RK_15 轮廓检测机构轮廓测量值开始字
ANDLD
ORLD
@SET W313.09  ; RK_15 轮廓检测机构#2移载#1点测量NG标志
LD TR1
LD W313.08  ; RK_15 轮廓检测机构#2移载#1点测量OK标志
ANDNOT W313.09  ; RK_15 轮廓检测机构#2移载#1点测量NG标志
LD W313.09  ; RK_15 轮廓检测机构#2移载#1点测量NG标志
ANDNOT W313.08  ; RK_15 轮廓检测机构#2移载#1点测量OK标志
ORLD
ANDLD
RSET W310.12  ; RK_15 轮廓检测机构#2移载#1轮廓测量值读取标志
RSET W314.06  ; RK_15 轮廓检测机构#2移载#1轮廓测量选择（手动）
LD TR0
AND W310.13  ; RK_15 轮廓检测机构#2移载#2轮廓测量值读取标志
OUT TR0
ANDNOT W311.13  ; RK_15 轮廓检测机构#2移载#2轮廓测量数据浮点数|字符显示标志（浮点数显示=0）
AND<>(305) #5858 D4426  ; RK_15 轮廓检测机构轮廓测量值开始字
AND<>(305) #2B46 D4426  ; RK_15 轮廓检测机构轮廓测量值开始字
AND<>(305) #2D46 D4426  ; RK_15 轮廓检测机构轮廓测量值开始字
OUT TR1
AND<F(331) D2312 D2210  ; RK_15 轮廓检测机构#2移载#2轮廓测量值（Float）, RK_15 轮廓检测机构#2移载轮廓测量值上限（Float）
AND>F(333) D2312 D2212  ; RK_15 轮廓检测机构#2移载#2轮廓测量值（Float）, RK_15 轮廓检测机构#2移载轮廓测量值下限（Float）
@SET W313.10  ; RK_15 轮廓检测机构#2移载#2点测量OK标志
LD TR1
LD>=F(334) D2312 D2210  ; RK_15 轮廓检测机构#2移载#2轮廓测量值（Float）, RK_15 轮廓检测机构#2移载轮廓测量值上限（Float）
OR<=F(332) D2312 D2212  ; RK_15 轮廓检测机构#2移载#2轮廓测量值（Float）, RK_15 轮廓检测机构#2移载轮廓测量值下限（Float）
ANDLD
LD TR0
AND W311.13  ; RK_15 轮廓检测机构#2移载#2轮廓测量数据浮点数|字符显示标志（浮点数显示=0）
LD=(300) #5858 D4426  ; RK_15 轮廓检测机构轮廓测量值开始字
OR=(300) #2B46 D4426  ; RK_15 轮廓检测机构轮廓测量值开始字
OR=(300) #2D46 D4426  ; RK_15 轮廓检测机构轮廓测量值开始字
ANDLD
ORLD
@SET W313.11  ; RK_15 轮廓检测机构#2移载#2点测量NG标志
LD TR0
LD W313.10  ; RK_15 轮廓检测机构#2移载#2点测量OK标志
ANDNOT W313.11  ; RK_15 轮廓检测机构#2移载#2点测量NG标志
LD W313.11  ; RK_15 轮廓检测机构#2移载#2点测量NG标志
ANDNOT W313.10  ; RK_15 轮廓检测机构#2移载#2点测量OK标志
ORLD
ANDLD
RSET W310.13  ; RK_15 轮廓检测机构#2移载#2轮廓测量值读取标志
RSET W314.07  ; RK_15 轮廓检测机构#2移载#2轮廓测量选择（手动）

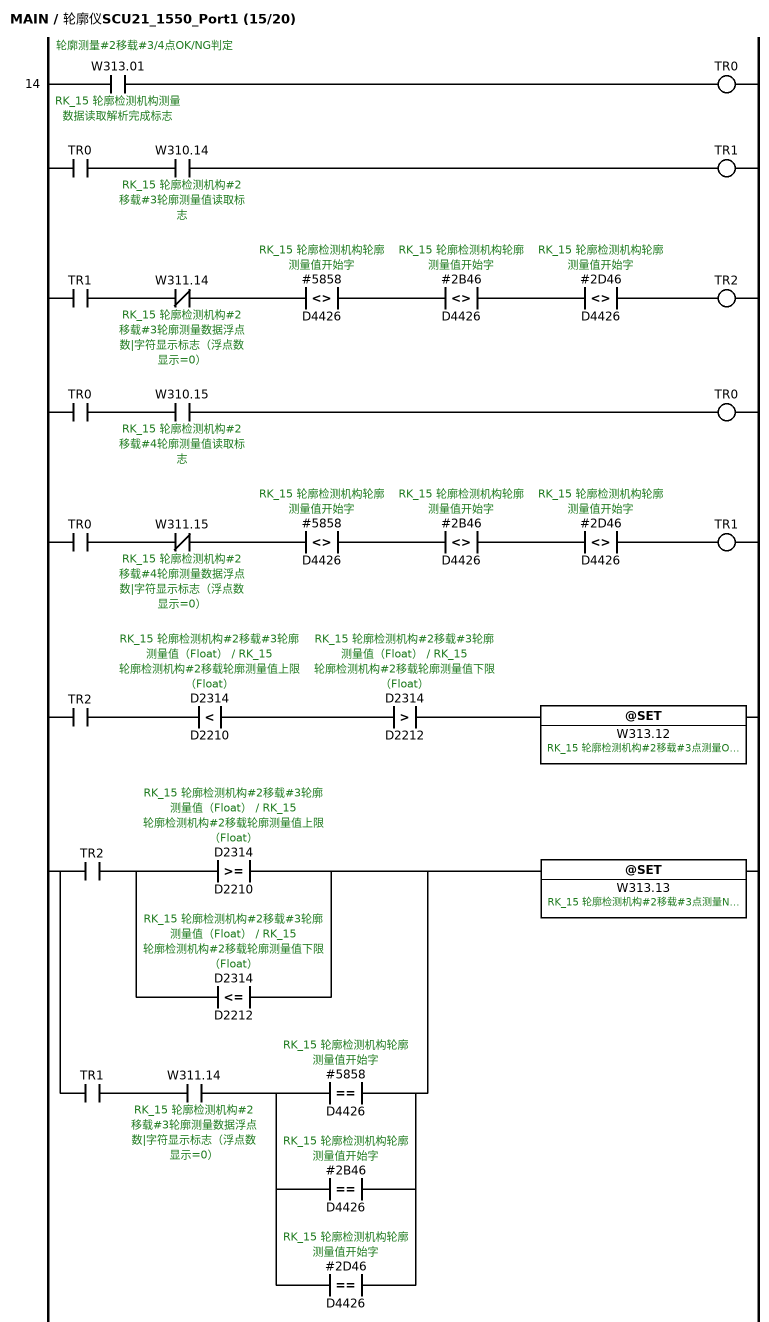

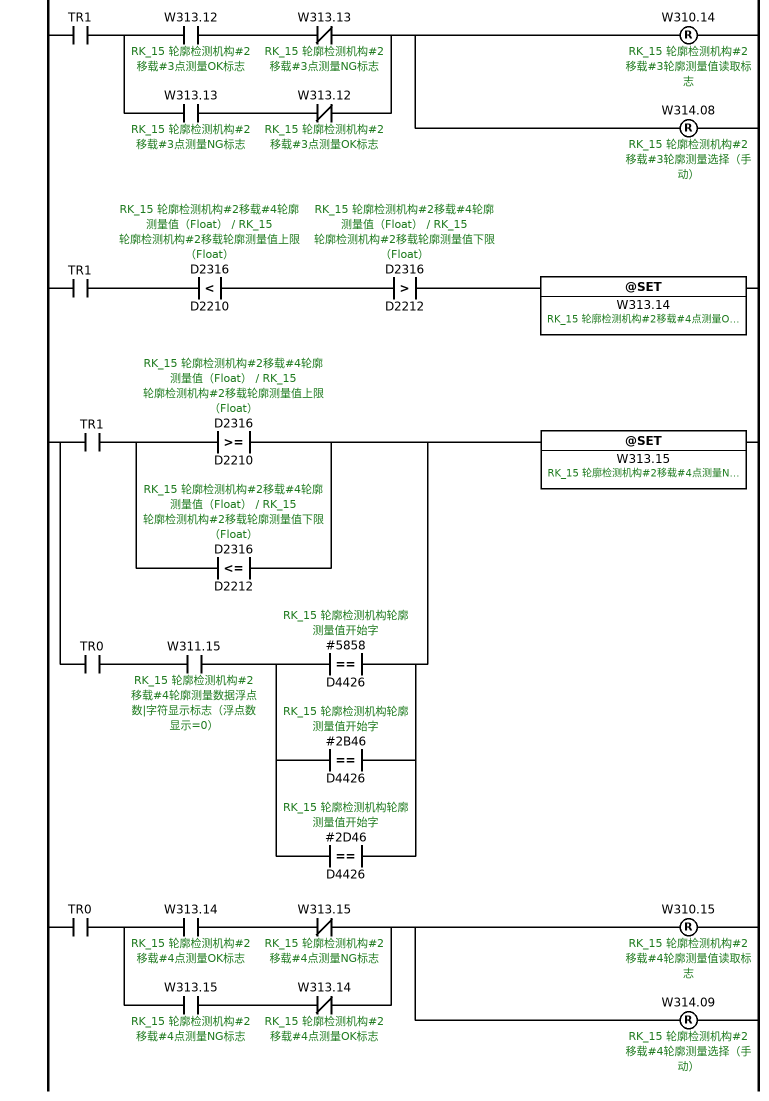
; rung 14: 轮廓测量#2移载#3/4点OK/NG判定
LD W313.01  ; RK_15 轮廓检测机构测量数据读取解析完成标志
OUT TR0
AND W310.14  ; RK_15 轮廓检测机构#2移载#3轮廓测量值读取标志
OUT TR1
ANDNOT W311.14  ; RK_15 轮廓检测机构#2移载#3轮廓测量数据浮点数|字符显示标志（浮点数显示=0）
AND<>(305) #5858 D4426  ; RK_15 轮廓检测机构轮廓测量值开始字
AND<>(305) #2B46 D4426  ; RK_15 轮廓检测机构轮廓测量值开始字
AND<>(305) #2D46 D4426  ; RK_15 轮廓检测机构轮廓测量值开始字
OUT TR2
AND<F(331) D2314 D2210  ; RK_15 轮廓检测机构#2移载#3轮廓测量值（Float）, RK_15 轮廓检测机构#2移载轮廓测量值上限（Float）
AND>F(333) D2314 D2212  ; RK_15 轮廓检测机构#2移载#3轮廓测量值（Float）, RK_15 轮廓检测机构#2移载轮廓测量值下限（Float）
@SET W313.12  ; RK_15 轮廓检测机构#2移载#3点测量OK标志
LD TR2
LD>=F(334) D2314 D2210  ; RK_15 轮廓检测机构#2移载#3轮廓测量值（Float）, RK_15 轮廓检测机构#2移载轮廓测量值上限（Float）
OR<=F(332) D2314 D2212  ; RK_15 轮廓检测机构#2移载#3轮廓测量值（Float）, RK_15 轮廓检测机构#2移载轮廓测量值下限（Float）
ANDLD
LD TR1
AND W311.14  ; RK_15 轮廓检测机构#2移载#3轮廓测量数据浮点数|字符显示标志（浮点数显示=0）
LD=(300) #5858 D4426  ; RK_15 轮廓检测机构轮廓测量值开始字
OR=(300) #2B46 D4426  ; RK_15 轮廓检测机构轮廓测量值开始字
OR=(300) #2D46 D4426  ; RK_15 轮廓检测机构轮廓测量值开始字
ANDLD
ORLD
@SET W313.13  ; RK_15 轮廓检测机构#2移载#3点测量NG标志
LD TR1
LD W313.12  ; RK_15 轮廓检测机构#2移载#3点测量OK标志
ANDNOT W313.13  ; RK_15 轮廓检测机构#2移载#3点测量NG标志
LD W313.13  ; RK_15 轮廓检测机构#2移载#3点测量NG标志
ANDNOT W313.12  ; RK_15 轮廓检测机构#2移载#3点测量OK标志
ORLD
ANDLD
RSET W310.14  ; RK_15 轮廓检测机构#2移载#3轮廓测量值读取标志
RSET W314.08  ; RK_15 轮廓检测机构#2移载#3轮廓测量选择（手动）
LD TR0
AND W310.15  ; RK_15 轮廓检测机构#2移载#4轮廓测量值读取标志
OUT TR0
ANDNOT W311.15  ; RK_15 轮廓检测机构#2移载#4轮廓测量数据浮点数|字符显示标志（浮点数显示=0）
AND<>(305) #5858 D4426  ; RK_15 轮廓检测机构轮廓测量值开始字
AND<>(305) #2B46 D4426  ; RK_15 轮廓检测机构轮廓测量值开始字
AND<>(305) #2D46 D4426  ; RK_15 轮廓检测机构轮廓测量值开始字
OUT TR1
AND<F(331) D2316 D2210  ; RK_15 轮廓检测机构#2移载#4轮廓测量值（Float）, RK_15 轮廓检测机构#2移载轮廓测量值上限（Float）
AND>F(333) D2316 D2212  ; RK_15 轮廓检测机构#2移载#4轮廓测量值（Float）, RK_15 轮廓检测机构#2移载轮廓测量值下限（Float）
@SET W313.14  ; RK_15 轮廓检测机构#2移载#4点测量OK标志
LD TR1
LD>=F(334) D2316 D2210  ; RK_15 轮廓检测机构#2移载#4轮廓测量值（Float）, RK_15 轮廓检测机构#2移载轮廓测量值上限（Float）
OR<=F(332) D2316 D2212  ; RK_15 轮廓检测机构#2移载#4轮廓测量值（Float）, RK_15 轮廓检测机构#2移载轮廓测量值下限（Float）
ANDLD
LD TR0
AND W311.15  ; RK_15 轮廓检测机构#2移载#4轮廓测量数据浮点数|字符显示标志（浮点数显示=0）
LD=(300) #5858 D4426  ; RK_15 轮廓检测机构轮廓测量值开始字
OR=(300) #2B46 D4426  ; RK_15 轮廓检测机构轮廓测量值开始字
OR=(300) #2D46 D4426  ; RK_15 轮廓检测机构轮廓测量值开始字
ANDLD
ORLD
@SET W313.15  ; RK_15 轮廓检测机构#2移载#4点测量NG标志
LD TR0
LD W313.14  ; RK_15 轮廓检测机构#2移载#4点测量OK标志
ANDNOT W313.15  ; RK_15 轮廓检测机构#2移载#4点测量NG标志
LD W313.15  ; RK_15 轮廓检测机构#2移载#4点测量NG标志
ANDNOT W313.14  ; RK_15 轮廓检测机构#2移载#4点测量OK标志
ORLD
ANDLD
RSET W310.15  ; RK_15 轮廓检测机构#2移载#4轮廓测量值读取标志
RSET W314.09  ; RK_15 轮廓检测机构#2移载#4轮廓测量选择（手动）

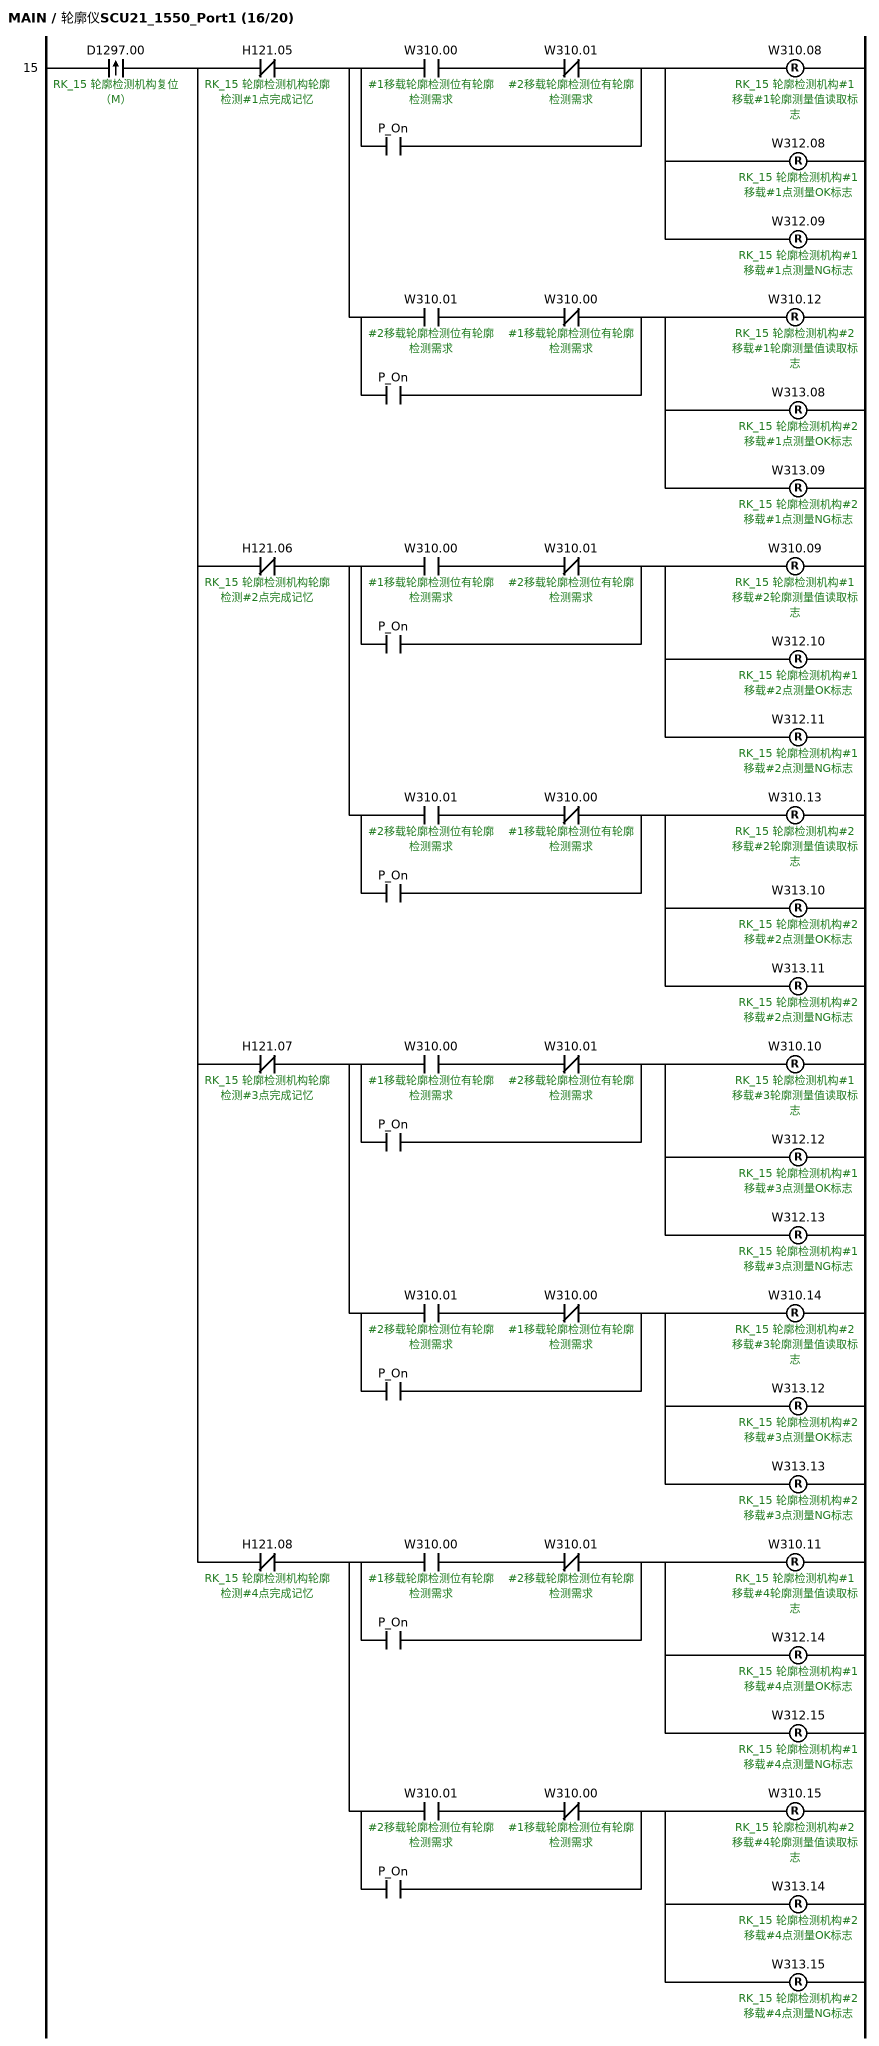
; rung 15
@LD D1297.00  ; RK_15 轮廓检测机构复位（M）
OUT TR0
ANDNOT H121.05  ; RK_15 轮廓检测机构轮廓检测#1点完成记忆
OUT TR1
LD W310.00  ; #1移载轮廓检测位有轮廓检测需求
ANDNOT W310.01  ; #2移载轮廓检测位有轮廓检测需求
OR P_On
ANDLD
RSET W310.08  ; RK_15 轮廓检测机构#1移载#1轮廓测量值读取标志
RSET W312.08  ; RK_15 轮廓检测机构#1移载#1点测量OK标志
RSET W312.09  ; RK_15 轮廓检测机构#1移载#1点测量NG标志
LD TR1
LD W310.01  ; #2移载轮廓检测位有轮廓检测需求
ANDNOT W310.00  ; #1移载轮廓检测位有轮廓检测需求
OR P_On
ANDLD
RSET W310.12  ; RK_15 轮廓检测机构#2移载#1轮廓测量值读取标志
RSET W313.08  ; RK_15 轮廓检测机构#2移载#1点测量OK标志
RSET W313.09  ; RK_15 轮廓检测机构#2移载#1点测量NG标志
LD TR0
ANDNOT H121.06  ; RK_15 轮廓检测机构轮廓检测#2点完成记忆
OUT TR1
LD W310.00  ; #1移载轮廓检测位有轮廓检测需求
ANDNOT W310.01  ; #2移载轮廓检测位有轮廓检测需求
OR P_On
ANDLD
RSET W310.09  ; RK_15 轮廓检测机构#1移载#2轮廓测量值读取标志
RSET W312.10  ; RK_15 轮廓检测机构#1移载#2点测量OK标志
RSET W312.11  ; RK_15 轮廓检测机构#1移载#2点测量NG标志
LD TR1
LD W310.01  ; #2移载轮廓检测位有轮廓检测需求
ANDNOT W310.00  ; #1移载轮廓检测位有轮廓检测需求
OR P_On
ANDLD
RSET W310.13  ; RK_15 轮廓检测机构#2移载#2轮廓测量值读取标志
RSET W313.10  ; RK_15 轮廓检测机构#2移载#2点测量OK标志
RSET W313.11  ; RK_15 轮廓检测机构#2移载#2点测量NG标志
LD TR0
ANDNOT H121.07  ; RK_15 轮廓检测机构轮廓检测#3点完成记忆
OUT TR1
LD W310.00  ; #1移载轮廓检测位有轮廓检测需求
ANDNOT W310.01  ; #2移载轮廓检测位有轮廓检测需求
OR P_On
ANDLD
RSET W310.10  ; RK_15 轮廓检测机构#1移载#3轮廓测量值读取标志
RSET W312.12  ; RK_15 轮廓检测机构#1移载#3点测量OK标志
RSET W312.13  ; RK_15 轮廓检测机构#1移载#3点测量NG标志
LD TR1
LD W310.01  ; #2移载轮廓检测位有轮廓检测需求
ANDNOT W310.00  ; #1移载轮廓检测位有轮廓检测需求
OR P_On
ANDLD
RSET W310.14  ; RK_15 轮廓检测机构#2移载#3轮廓测量值读取标志
RSET W313.12  ; RK_15 轮廓检测机构#2移载#3点测量OK标志
RSET W313.13  ; RK_15 轮廓检测机构#2移载#3点测量NG标志
LD TR0
ANDNOT H121.08  ; RK_15 轮廓检测机构轮廓检测#4点完成记忆
OUT TR0
LD W310.00  ; #1移载轮廓检测位有轮廓检测需求
ANDNOT W310.01  ; #2移载轮廓检测位有轮廓检测需求
OR P_On
ANDLD
RSET W310.11  ; RK_15 轮廓检测机构#1移载#4轮廓测量值读取标志
RSET W312.14  ; RK_15 轮廓检测机构#1移载#4点测量OK标志
RSET W312.15  ; RK_15 轮廓检测机构#1移载#4点测量NG标志
LD TR0
LD W310.01  ; #2移载轮廓检测位有轮廓检测需求
ANDNOT W310.00  ; #1移载轮廓检测位有轮廓检测需求
OR P_On
ANDLD
RSET W310.15  ; RK_15 轮廓检测机构#2移载#4轮廓测量值读取标志
RSET W313.14  ; RK_15 轮廓检测机构#2移载#4点测量OK标志
RSET W313.15  ; RK_15 轮廓检测机构#2移载#4点测量NG标志

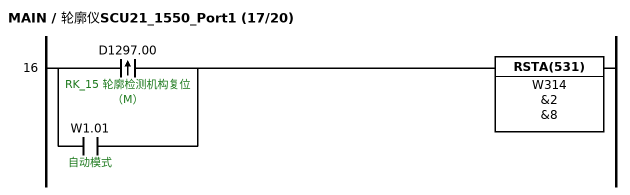
; rung 16
@LD D1297.00  ; RK_15 轮廓检测机构复位（M）
OR W1.01  ; 自动模式
RSTA(531) W314 &2 &8

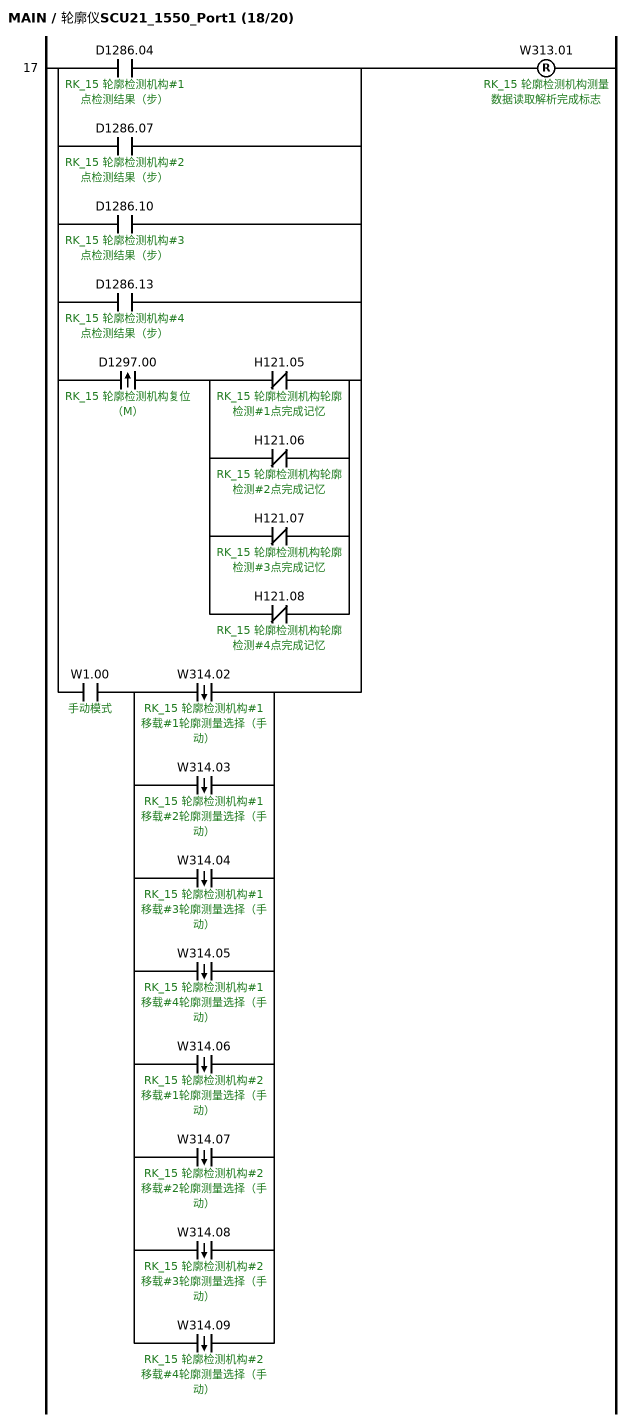
; rung 17
LD D1286.04  ; RK_15 轮廓检测机构#1点检测结果（步）
OR D1286.07  ; RK_15 轮廓检测机构#2点检测结果（步）
OR D1286.10  ; RK_15 轮廓检测机构#3点检测结果（步）
OR D1286.13  ; RK_15 轮廓检测机构#4点检测结果（步）
@LD D1297.00  ; RK_15 轮廓检测机构复位（M）
LDNOT H121.05  ; RK_15 轮廓检测机构轮廓检测#1点完成记忆
ORNOT H121.06  ; RK_15 轮廓检测机构轮廓检测#2点完成记忆
ORNOT H121.07  ; RK_15 轮廓检测机构轮廓检测#3点完成记忆
ORNOT H121.08  ; RK_15 轮廓检测机构轮廓检测#4点完成记忆
ANDLD
ORLD
LD W1.00  ; 手动模式
%LD W314.02  ; RK_15 轮廓检测机构#1移载#1轮廓测量选择（手动）
%OR W314.03  ; RK_15 轮廓检测机构#1移载#2轮廓测量选择（手动）
%OR W314.04  ; RK_15 轮廓检测机构#1移载#3轮廓测量选择（手动）
%OR W314.05  ; RK_15 轮廓检测机构#1移载#4轮廓测量选择（手动）
%OR W314.06  ; RK_15 轮廓检测机构#2移载#1轮廓测量选择（手动）
%OR W314.07  ; RK_15 轮廓检测机构#2移载#2轮廓测量选择（手动）
%OR W314.08  ; RK_15 轮廓检测机构#2移载#3轮廓测量选择（手动）
%OR W314.09  ; RK_15 轮廓检测机构#2移载#4轮廓测量选择（手动）
ANDLD
ORLD
RSET W313.01  ; RK_15 轮廓检测机构测量数据读取解析完成标志

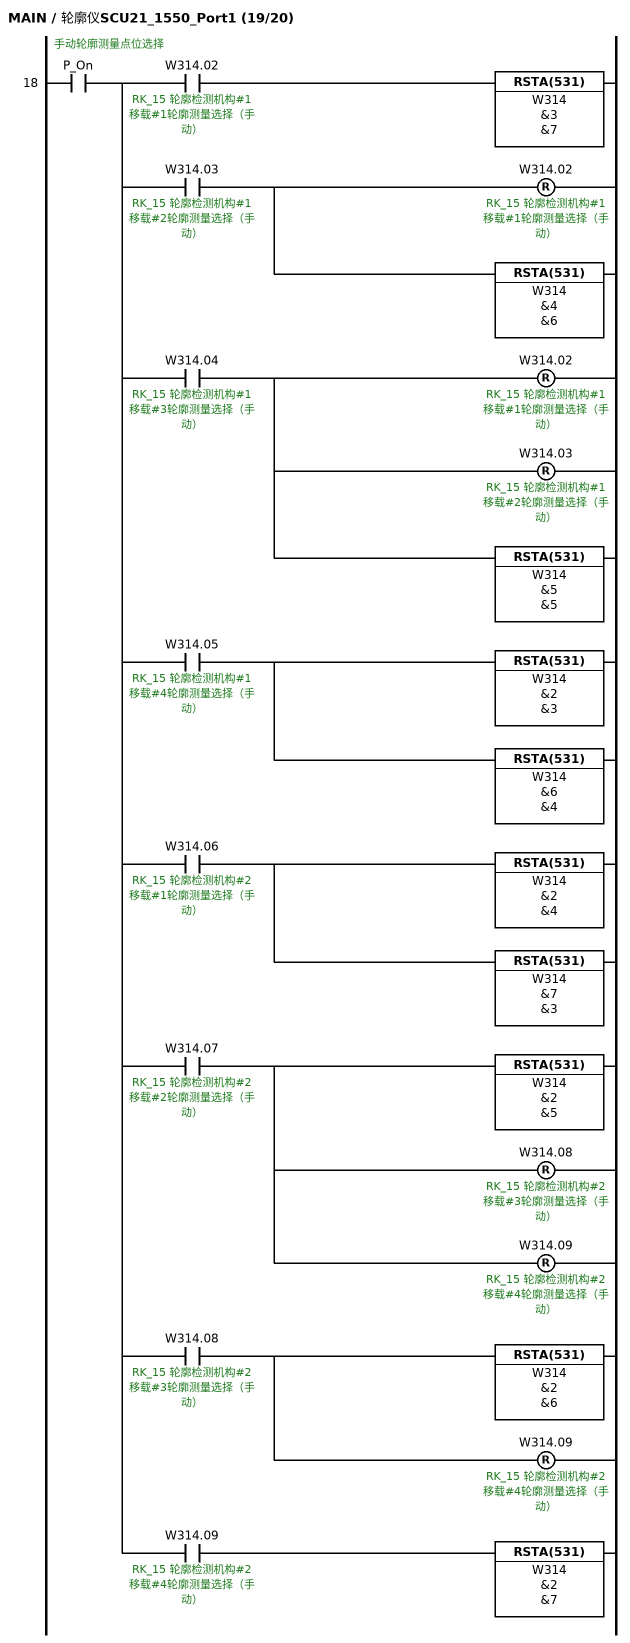
; rung 18: 手动轮廓测量点位选择
LD P_On
OUT TR0
AND W314.02  ; RK_15 轮廓检测机构#1移载#1轮廓测量选择（手动）
RSTA(531) W314 &3 &7
LD TR0
AND W314.03  ; RK_15 轮廓检测机构#1移载#2轮廓测量选择（手动）
RSET W314.02  ; RK_15 轮廓检测机构#1移载#1轮廓测量选择（手动）
RSTA(531) W314 &4 &6
LD TR0
AND W314.04  ; RK_15 轮廓检测机构#1移载#3轮廓测量选择（手动）
RSET W314.02  ; RK_15 轮廓检测机构#1移载#1轮廓测量选择（手动）
RSET W314.03  ; RK_15 轮廓检测机构#1移载#2轮廓测量选择（手动）
RSTA(531) W314 &5 &5
LD TR0
AND W314.05  ; RK_15 轮廓检测机构#1移载#4轮廓测量选择（手动）
RSTA(531) W314 &2 &3
RSTA(531) W314 &6 &4
LD TR0
AND W314.06  ; RK_15 轮廓检测机构#2移载#1轮廓测量选择（手动）
RSTA(531) W314 &2 &4
RSTA(531) W314 &7 &3
LD TR0
AND W314.07  ; RK_15 轮廓检测机构#2移载#2轮廓测量选择（手动）
RSTA(531) W314 &2 &5
RSET W314.08  ; RK_15 轮廓检测机构#2移载#3轮廓测量选择（手动）
RSET W314.09  ; RK_15 轮廓检测机构#2移载#4轮廓测量选择（手动）
LD TR0
AND W314.08  ; RK_15 轮廓检测机构#2移载#3轮廓测量选择（手动）
RSTA(531) W314 &2 &6
RSET W314.09  ; RK_15 轮廓检测机构#2移载#4轮廓测量选择（手动）
LD TR0
AND W314.09  ; RK_15 轮廓检测机构#2移载#4轮廓测量选择（手动）
RSTA(531) W314 &2 &7

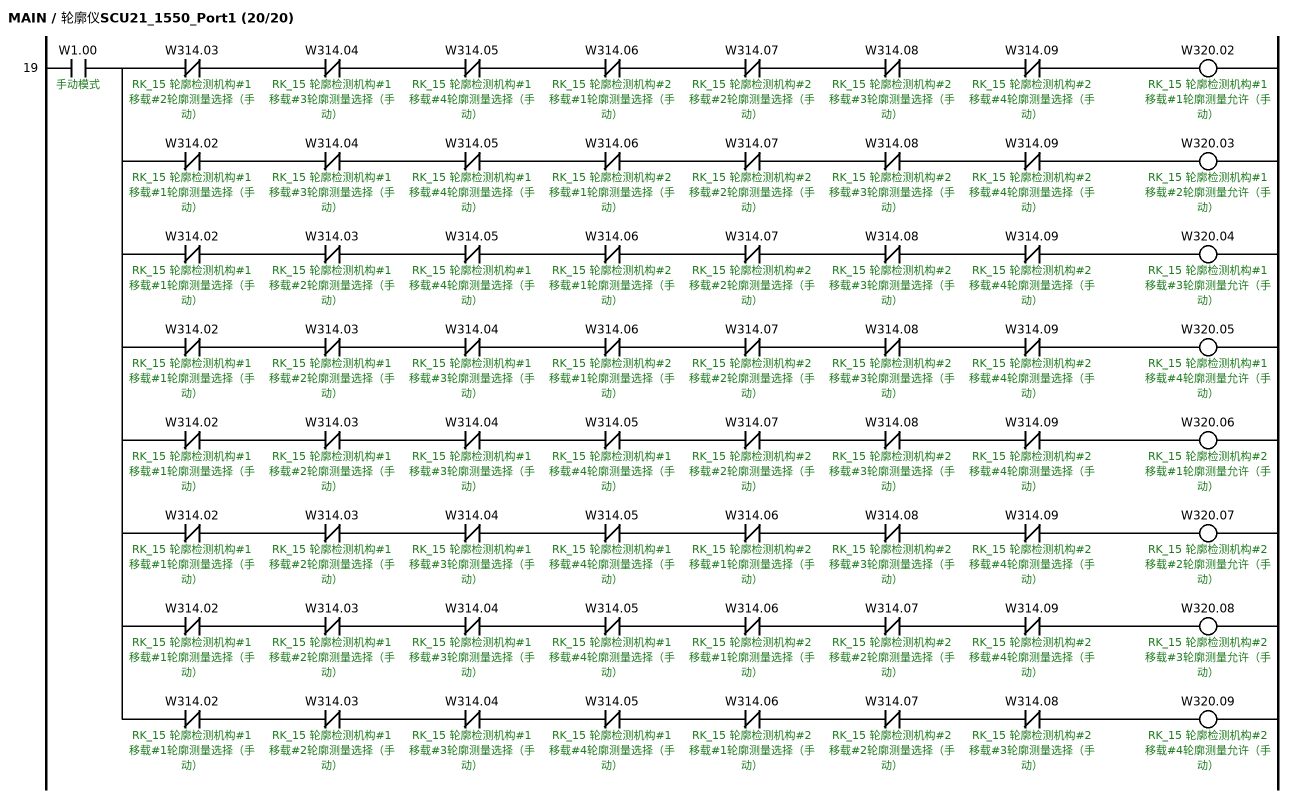
; rung 19
LD W1.00  ; 手动模式
OUT TR0
ANDNOT W314.03  ; RK_15 轮廓检测机构#1移载#2轮廓测量选择（手动）
ANDNOT W314.04  ; RK_15 轮廓检测机构#1移载#3轮廓测量选择（手动）
ANDNOT W314.05  ; RK_15 轮廓检测机构#1移载#4轮廓测量选择（手动）
ANDNOT W314.06  ; RK_15 轮廓检测机构#2移载#1轮廓测量选择（手动）
ANDNOT W314.07  ; RK_15 轮廓检测机构#2移载#2轮廓测量选择（手动）
ANDNOT W314.08  ; RK_15 轮廓检测机构#2移载#3轮廓测量选择（手动）
ANDNOT W314.09  ; RK_15 轮廓检测机构#2移载#4轮廓测量选择（手动）
OUT W320.02  ; RK_15 轮廓检测机构#1移载#1轮廓测量允许（手动）
LD TR0
ANDNOT W314.02  ; RK_15 轮廓检测机构#1移载#1轮廓测量选择（手动）
ANDNOT W314.04  ; RK_15 轮廓检测机构#1移载#3轮廓测量选择（手动）
ANDNOT W314.05  ; RK_15 轮廓检测机构#1移载#4轮廓测量选择（手动）
ANDNOT W314.06  ; RK_15 轮廓检测机构#2移载#1轮廓测量选择（手动）
ANDNOT W314.07  ; RK_15 轮廓检测机构#2移载#2轮廓测量选择（手动）
ANDNOT W314.08  ; RK_15 轮廓检测机构#2移载#3轮廓测量选择（手动）
ANDNOT W314.09  ; RK_15 轮廓检测机构#2移载#4轮廓测量选择（手动）
OUT W320.03  ; RK_15 轮廓检测机构#1移载#2轮廓测量允许（手动）
LD TR0
ANDNOT W314.02  ; RK_15 轮廓检测机构#1移载#1轮廓测量选择（手动）
ANDNOT W314.03  ; RK_15 轮廓检测机构#1移载#2轮廓测量选择（手动）
ANDNOT W314.05  ; RK_15 轮廓检测机构#1移载#4轮廓测量选择（手动）
ANDNOT W314.06  ; RK_15 轮廓检测机构#2移载#1轮廓测量选择（手动）
ANDNOT W314.07  ; RK_15 轮廓检测机构#2移载#2轮廓测量选择（手动）
ANDNOT W314.08  ; RK_15 轮廓检测机构#2移载#3轮廓测量选择（手动）
ANDNOT W314.09  ; RK_15 轮廓检测机构#2移载#4轮廓测量选择（手动）
OUT W320.04  ; RK_15 轮廓检测机构#1移载#3轮廓测量允许（手动）
LD TR0
ANDNOT W314.02  ; RK_15 轮廓检测机构#1移载#1轮廓测量选择（手动）
ANDNOT W314.03  ; RK_15 轮廓检测机构#1移载#2轮廓测量选择（手动）
ANDNOT W314.04  ; RK_15 轮廓检测机构#1移载#3轮廓测量选择（手动）
ANDNOT W314.06  ; RK_15 轮廓检测机构#2移载#1轮廓测量选择（手动）
ANDNOT W314.07  ; RK_15 轮廓检测机构#2移载#2轮廓测量选择（手动）
ANDNOT W314.08  ; RK_15 轮廓检测机构#2移载#3轮廓测量选择（手动）
ANDNOT W314.09  ; RK_15 轮廓检测机构#2移载#4轮廓测量选择（手动）
OUT W320.05  ; RK_15 轮廓检测机构#1移载#4轮廓测量允许（手动）
LD TR0
ANDNOT W314.02  ; RK_15 轮廓检测机构#1移载#1轮廓测量选择（手动）
ANDNOT W314.03  ; RK_15 轮廓检测机构#1移载#2轮廓测量选择（手动）
ANDNOT W314.04  ; RK_15 轮廓检测机构#1移载#3轮廓测量选择（手动）
ANDNOT W314.05  ; RK_15 轮廓检测机构#1移载#4轮廓测量选择（手动）
ANDNOT W314.07  ; RK_15 轮廓检测机构#2移载#2轮廓测量选择（手动）
ANDNOT W314.08  ; RK_15 轮廓检测机构#2移载#3轮廓测量选择（手动）
ANDNOT W314.09  ; RK_15 轮廓检测机构#2移载#4轮廓测量选择（手动）
OUT W320.06  ; RK_15 轮廓检测机构#2移载#1轮廓测量允许（手动）
LD TR0
ANDNOT W314.02  ; RK_15 轮廓检测机构#1移载#1轮廓测量选择（手动）
ANDNOT W314.03  ; RK_15 轮廓检测机构#1移载#2轮廓测量选择（手动）
ANDNOT W314.04  ; RK_15 轮廓检测机构#1移载#3轮廓测量选择（手动）
ANDNOT W314.05  ; RK_15 轮廓检测机构#1移载#4轮廓测量选择（手动）
ANDNOT W314.06  ; RK_15 轮廓检测机构#2移载#1轮廓测量选择（手动）
ANDNOT W314.08  ; RK_15 轮廓检测机构#2移载#3轮廓测量选择（手动）
ANDNOT W314.09  ; RK_15 轮廓检测机构#2移载#4轮廓测量选择（手动）
OUT W320.07  ; RK_15 轮廓检测机构#2移载#2轮廓测量允许（手动）
LD TR0
ANDNOT W314.02  ; RK_15 轮廓检测机构#1移载#1轮廓测量选择（手动）
ANDNOT W314.03  ; RK_15 轮廓检测机构#1移载#2轮廓测量选择（手动）
ANDNOT W314.04  ; RK_15 轮廓检测机构#1移载#3轮廓测量选择（手动）
ANDNOT W314.05  ; RK_15 轮廓检测机构#1移载#4轮廓测量选择（手动）
ANDNOT W314.06  ; RK_15 轮廓检测机构#2移载#1轮廓测量选择（手动）
ANDNOT W314.07  ; RK_15 轮廓检测机构#2移载#2轮廓测量选择（手动）
ANDNOT W314.09  ; RK_15 轮廓检测机构#2移载#4轮廓测量选择（手动）
OUT W320.08  ; RK_15 轮廓检测机构#2移载#3轮廓测量允许（手动）
LD TR0
ANDNOT W314.02  ; RK_15 轮廓检测机构#1移载#1轮廓测量选择（手动）
ANDNOT W314.03  ; RK_15 轮廓检测机构#1移载#2轮廓测量选择（手动）
ANDNOT W314.04  ; RK_15 轮廓检测机构#1移载#3轮廓测量选择（手动）
ANDNOT W314.05  ; RK_15 轮廓检测机构#1移载#4轮廓测量选择（手动）
ANDNOT W314.06  ; RK_15 轮廓检测机构#2移载#1轮廓测量选择（手动）
ANDNOT W314.07  ; RK_15 轮廓检测机构#2移载#2轮廓测量选择（手动）
ANDNOT W314.08  ; RK_15 轮廓检测机构#2移载#3轮廓测量选择（手动）
OUT W320.09  ; RK_15 轮廓检测机构#2移载#4轮廓测量允许（手动）

### Section Hipot检测SCU21_1550_Port2

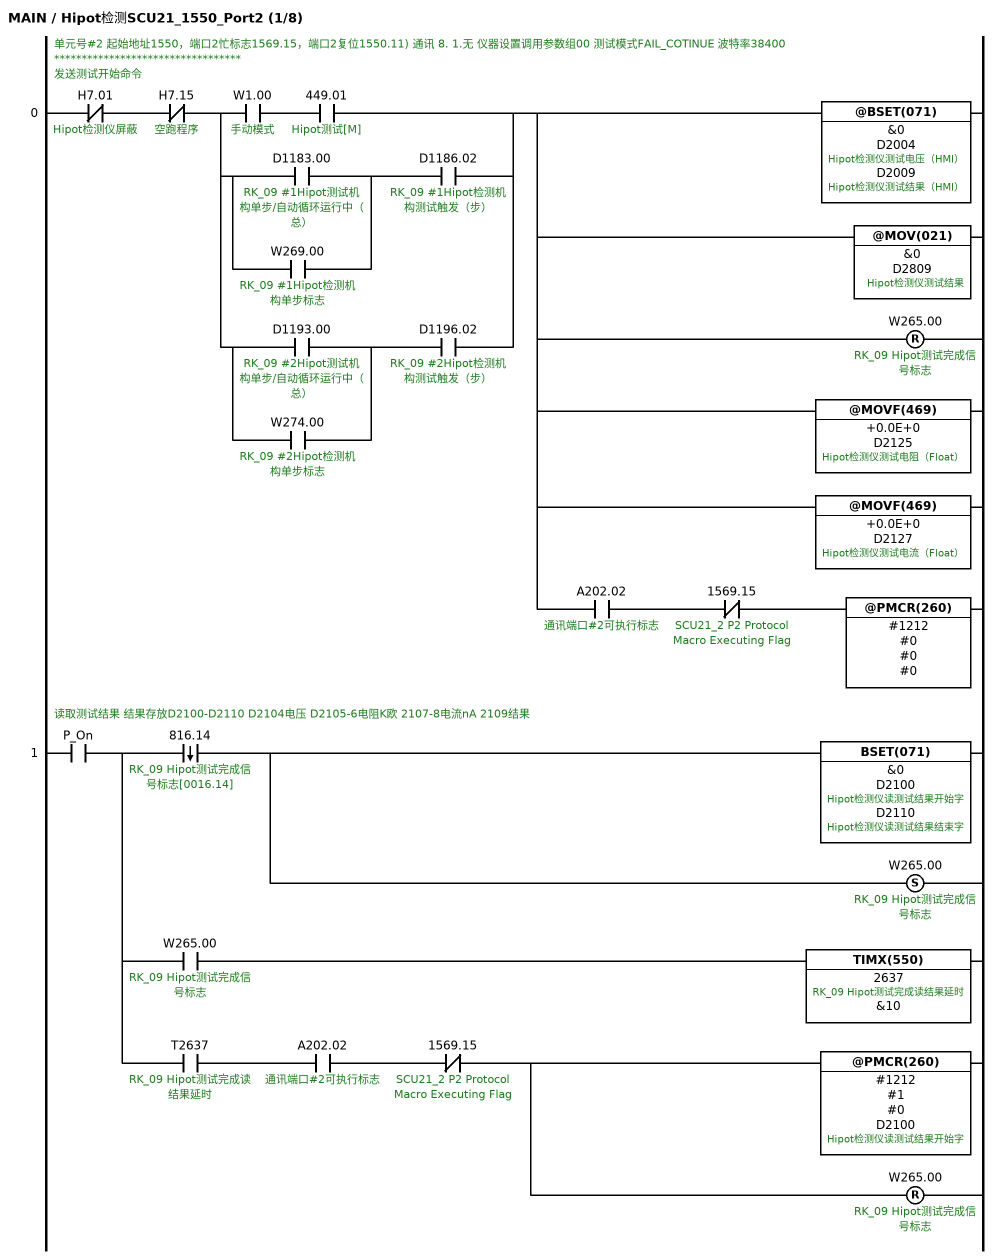
; rung 0: 单元号#2 起始地址1550，端口2忙标志1569.15，端口2复位1550.11) 通讯 8. 1.无 仪器设置调用参数组00 测试模式FAIL_COTINUE 波特率38400 / ********************************** / 发送测试开始命令
LDNOT H7.01  ; Hipot检测仪屏蔽
ANDNOT H7.15  ; 空跑程序
LD W1.00  ; 手动模式
AND 449.01  ; Hipot测试[M]
LD D1183.00  ; RK_09 #1Hipot测试机构单步/自动循环运行中（总）
OR W269.00  ; RK_09 #1Hipot检测机构单步标志
AND D1186.02  ; RK_09 #1Hipot检测机构测试触发（步）
ORLD
LD D1193.00  ; RK_09 #2Hipot测试机构单步/自动循环运行中（总）
OR W274.00  ; RK_09 #2Hipot检测机构单步标志
AND D1196.02  ; RK_09 #2Hipot检测机构测试触发（步）
ORLD
ANDLD
@BSET(071) &0 D2004 D2009  ; Hipot检测仪测试电压（HMI）, Hipot检测仪测试结果（HMI）
@MOV(021) &0 D2809  ; Hipot检测仪测试结果
RSET W265.00  ; RK_09 Hipot测试完成信号标志
@MOVF(469) +0.0E+0 D2125  ; Hipot检测仪测试电阻（Float）
@MOVF(469) +0.0E+0 D2127  ; Hipot检测仪测试电流（Float）
AND A202.02  ; 通讯端口#2可执行标志
ANDNOT 1569.15  ; SCU21_2 P2 Protocol Macro Executing Flag
@PMCR(260) #1212 #0 #0 #0
; rung 1: 读取测试结果 结果存放D2100-D2110 D2104电压 D2105-6电阻K欧 2107-8电流nA 2109结果
LD P_On
OUT TR0
%AND 816.14  ; RK_09 Hipot测试完成信号标志[0016.14]
BSET(071) &0 D2100 D2110  ; Hipot检测仪读测试结果开始字, Hipot检测仪读测试结果结束字
SET W265.00  ; RK_09 Hipot测试完成信号标志
LD TR0
AND W265.00  ; RK_09 Hipot测试完成信号标志
TIMX(550) 2637 &10  ; RK_09 Hipot测试完成读结果延时
LD TR0
AND T2637  ; RK_09 Hipot测试完成读结果延时
AND A202.02  ; 通讯端口#2可执行标志
ANDNOT 1569.15  ; SCU21_2 P2 Protocol Macro Executing Flag
@PMCR(260) #1212 #1 #0 D2100  ; Hipot检测仪读测试结果开始字
RSET W265.00  ; RK_09 Hipot测试完成信号标志

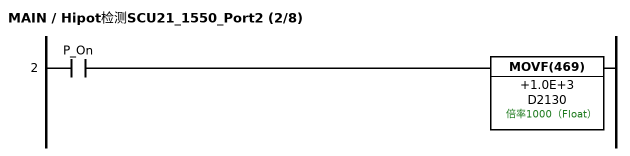
; rung 2
LD P_On
MOVF(469) +1.0E+3 D2130  ; 倍率1000（Float）

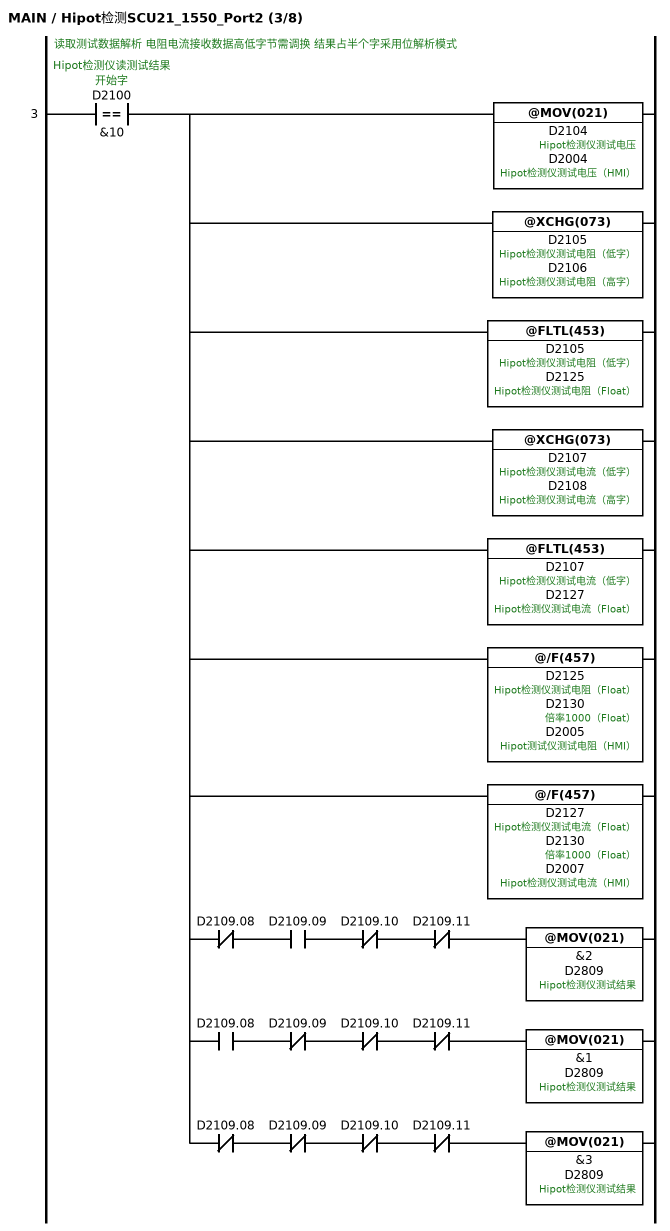
; rung 3: 读取测试数据解析 电阻电流接收数据高低字节需调换 结果占半个字采用位解析模式
LD=(300) D2100 &10  ; Hipot检测仪读测试结果开始字
OUT TR0
@MOV(021) D2104 D2004  ; Hipot检测仪测试电压, Hipot检测仪测试电压（HMI）
@XCHG(073) D2105 D2106  ; Hipot检测仪测试电阻（低字）, Hipot检测仪测试电阻（高字）
@FLTL(453) D2105 D2125  ; Hipot检测仪测试电阻（低字）, Hipot检测仪测试电阻（Float）
@XCHG(073) D2107 D2108  ; Hipot检测仪测试电流（低字）, Hipot检测仪测试电流（高字）
@FLTL(453) D2107 D2127  ; Hipot检测仪测试电流（低字）, Hipot检测仪测试电流（Float）
@/F(457) D2125 D2130 D2005  ; Hipot检测仪测试电阻（Float）, 倍率1000（Float）, Hipot测试仪测试电阻（HMI）  // KΩ→MΩ
@/F(457) D2127 D2130 D2007  ; Hipot检测仪测试电流（Float）, 倍率1000（Float）, Hipot检测仪测试电流（HMI）  // nA→uA
ANDNOT D2109.08
AND D2109.09
ANDNOT D2109.10
ANDNOT D2109.11
@MOV(021) &2 D2809  ; Hipot检测仪测试结果  // 2=NG
LD TR0
AND D2109.08
ANDNOT D2109.09
ANDNOT D2109.10
ANDNOT D2109.11
@MOV(021) &1 D2809  ; Hipot检测仪测试结果  // 1=OK
LD TR0
ANDNOT D2109.08
ANDNOT D2109.09
ANDNOT D2109.10
ANDNOT D2109.11
@MOV(021) &3 D2809  ; Hipot检测仪测试结果  // 3=无测试结果

